(*
version 1.1		06. apr 2011
programmer		ks
tested by			ks

TN_SELECT_TEXT dient zur verwaltung und darstellung einer Elementeauswahl
*)
(* Benutzereingabe auswerten -> Selektion Text n *)
IF Xus_TN_INPUT_CONTROL_DATA.bo_Focus = TRUE THEN

(* Leertaste-Taste auswerten *)
	IF Xus_TN_INPUT_CONTROL_DATA.by_Input_ASCII_Code = BYTE#32 THEN
		Xus_TN_INPUT_CONTROL_DATA.in_selected := Xus_TN_INPUT_CONTROL_DATA.in_selected + INT#01; 
		Xus_TN_INPUT_CONTROL_DATA.bo_Update_Input := TRUE;
	END_IF;
 
	(* Return-Taste auswerten *)
	IF Xus_TN_INPUT_CONTROL_DATA.by_Input_Exten_Code = BYTE#13 THEN
		Xus_TN_INPUT_CONTROL_DATA.bo_Input_Entered := TRUE;
	END_IF;

END_IF;

(* Aktualisierung der Anzeige *)
IF (Xus_TN_INPUT_CONTROL_DATA.bo_Update_Input = TRUE) OR (Xus_TN_INPUT_CONTROL_DATA.bo_Update_All = TRUE) THEN

	(* Title-Text ausgeben *)
	IF Xus_TN_INPUT_CONTROL_DATA.bo_Update_All = TRUE THEN

		IF (Xus_TN_INPUT_CONTROL_DATA.in_Title_X_Offset = INT#00) AND (Xus_TN_INPUT_CONTROL_DATA.in_Title_Y_Offset = INT#00) THEN
			(* wenn Offset X,Y =0 dann Titlestring links vom Element positionieren *)
			FB_TN_SC_WRITE.Iin_Y := Xus_TN_INPUT_CONTROL_DATA.in_Y;
			FB_TN_SC_WRITE.Iin_X := Xus_TN_INPUT_CONTROL_DATA.in_X - LEN(Xus_TN_INPUT_CONTROL_DATA.st_Title_String);

		ELSE
			(* Title-Text durch Row, Color-Offset ausgeben *)
			FB_TN_SC_WRITE.Iin_Y := Xus_TN_INPUT_CONTROL_DATA.in_Y + Xus_TN_INPUT_CONTROL_DATA.in_Title_Y_Offset;
			FB_TN_SC_WRITE.Iin_X := Xus_TN_INPUT_CONTROL_DATA.in_X + Xus_TN_INPUT_CONTROL_DATA.in_Title_X_Offset;
		END_IF;

		(* Title-Text durch Row, Color-Offset ausgeben *)
		FB_TN_SC_WRITE(	Iby_ATTR := Xus_TN_INPUT_CONTROL_DATA.by_Title_Attr,
						Ist_STRING := Xus_TN_INPUT_CONTROL_DATA.st_Title_String,
						Xus_TN_SCREEN := Xus_TN_SCREEN);

	END_IF;

	(* Eingabezeile verarbeiten *)

	(* Anzahl der Elemente bestimmen *)
	in_count := ELEMENT_COUNT(SEP:=BYTE#35,ELEMENT:=Xus_TN_INPUT_CONTROL_DATA.st_Input_Data);

	IF in_Count > INT#00 THEN

		IF Xus_TN_INPUT_CONTROL_DATA.in_selected < INT#1 THEN
			Xus_TN_INPUT_CONTROL_DATA.in_selected := INT#01;
		END_IF;

		IF Xus_TN_INPUT_CONTROL_DATA.in_selected > in_count THEN
			Xus_TN_INPUT_CONTROL_DATA.in_selected := INT#01;
		END_IF;

		st_String := ELEMENT_GET(SEP:=BYTE#35,POS:=Xus_TN_INPUT_CONTROL_DATA.in_selected - 1,ELEMENT:=Xus_TN_INPUT_CONTROL_DATA.st_Input_Data);

		st_String := FIX(	str:=st_String,
							L:=LEN(Xus_TN_INPUT_CONTROL_DATA.st_Input_Mask),
							C:=BYTE#32,
							M:=Xus_TN_INPUT_CONTROL_DATA.in_Input_Option);

		Xus_TN_INPUT_CONTROL_DATA.st_Input_String := st_String;

		IF Xus_TN_INPUT_CONTROL_DATA.bo_Focus = TRUE THEN
			by_Attr := Xus_TN_INPUT_CONTROL_DATA.by_Attr_mF;
		ELSE
			by_Attr := Xus_TN_INPUT_CONTROL_DATA.by_Attr_oF;
		END_IF;

		FB_TN_SC_WRITE(	Iin_Y := Xus_TN_INPUT_CONTROL_DATA.in_Y,
						Iin_X := Xus_TN_INPUT_CONTROL_DATA.in_X,
						Iby_ATTR := by_Attr,
						Ist_STRING := st_String,
						Xus_TN_SCREEN := Xus_TN_SCREEN);
	END_IF;

	(* Cursor auf aktuelle Position setzen *)
	Xus_TN_INPUT_CONTROL_DATA.in_Cursor_Y := Xus_TN_INPUT_CONTROL_DATA.in_Y;
	Xus_TN_INPUT_CONTROL_DATA.in_Cursor_X := Xus_TN_INPUT_CONTROL_DATA.in_X;

	(* Update-Flag's rücksetzen *)
	Xus_TN_INPUT_CONTROL_DATA.bo_Update_All := FALSE;
	Xus_TN_INPUT_CONTROL_DATA.bo_Update_Input := FALSE;

END_IF;

(* revision history

ks	06. apr. 2011	rev 1.1
	list_len und list_get durch element_count und element_get ersetzt

ks	10. mai. 2010	rev 1.0
	original version
*)
END_FUNCTION_BLOCK

(* POU TN_INPUT_EDIT_LINE, ST *)
FUNCTION_BLOCK TN_INPUT_EDIT_LINE
VAR
	in_count : INT;
	in_Count_End : INT;
	in_CursorOffset : INT;
	by_Attr : BYTE;
	st_String : STRING;
	bo_Pos_Found : BOOL;
	st_CHAR : STRING(1);
	in_old_charpos : INT;
END_VAR
VAR
	FB_TN_SC_WRITE : TN_SC_WRITE;
END_VAR
VAR_IN_OUT
	Xus_TN_SCREEN : us_TN_SCREEN;
	Xus_TN_INPUT_CONTROL_DATA : us_TN_INPUT_CONTROL_DATA;
END_VAR

(*
version 1.0		10. mai 2010
programmer		ks
tested by		ks

TN_INPUT_EDIT_LINE ermöglicht die Eingabe von Texten durch eine Editierbare Eingabezeile
*)
(* Cursorsteuerung rücksetzen *)
in_CursorOffset := INT#0;

IF Xus_TN_INPUT_CONTROL_DATA.bo_Focus = TRUE THEN

	(* Texteingabe erkannt ? *)
	IF Xus_TN_INPUT_CONTROL_DATA.by_Input_ASCII_Code > BYTE#0 THEN

		IF (Xus_TN_INPUT_CONTROL_DATA.bo_Input_Only_Num = TRUE AND Xus_TN_INPUT_CONTROL_DATA.bo_Input_ASCII_IsNum = TRUE)
			OR (Xus_TN_INPUT_CONTROL_DATA.bo_Input_Only_Num = FALSE) THEN

			(* ASCII Wert in einen String wandeln *)
			st_CHAR := CHR_TO_STRING(C:=Xus_TN_INPUT_CONTROL_DATA.by_Input_ASCII_Code);

			(* Eingabe übernehmen *)
			Xus_TN_INPUT_CONTROL_DATA.st_Input_Data := REPLACE(Xus_TN_INPUT_CONTROL_DATA.st_Input_Data,
			st_CHAR,INT#1,Xus_TN_INPUT_CONTROL_DATA.in_Cursor_Pos);

			in_CursorOffset := INT#1;
			Xus_TN_INPUT_CONTROL_DATA.bo_Update_Input := TRUE;
		END_IF;
	END_IF;

	CASE BYTE_TO_INT(Xus_TN_INPUT_CONTROL_DATA.by_Input_Exten_Code) OF

	67: (* Cursor rechts gedrückt *)
		in_CursorOffset := INT#1;

	68: (* Cursor links gedrückt *)
		in_CursorOffset := -1;

	08: (* Backspace gedrückt *)
		Xus_TN_INPUT_CONTROL_DATA.st_Input_Data := REPLACE(Xus_TN_INPUT_CONTROL_DATA.st_Input_Data, ' ', 1,Xus_TN_INPUT_CONTROL_DATA.in_Cursor_Pos);
		Xus_TN_INPUT_CONTROL_DATA.bo_Update_Input := TRUE;
		in_CursorOffset := -1;

	13: (* Enter-Taste gedrückt *)
		IF LEN(Xus_TN_INPUT_CONTROL_DATA.st_Input_Mask) > INT#00 THEN
			(* Eingabestring übernehmen *)
			Xus_TN_INPUT_CONTROL_DATA.st_Input_String := Xus_TN_INPUT_CONTROL_DATA.st_Input_Data;

			(* Eingabestring -> links und rechts Leerzeichen entfernen *)
			Xus_TN_INPUT_CONTROL_DATA.st_Input_String := TRIME(str:=Xus_TN_INPUT_CONTROL_DATA.st_Input_String);
			Xus_TN_INPUT_CONTROL_DATA.bo_Input_Entered := TRUE;

			(* neue Eingabe vorbereiten *)
			Xus_TN_INPUT_CONTROL_DATA.st_Input_Data := Xus_TN_INPUT_CONTROL_DATA.st_Input_Mask;

			Xus_TN_INPUT_CONTROL_DATA.in_Cursor_Pos := INT#1;
			Xus_TN_INPUT_CONTROL_DATA.bo_Update_Input := TRUE;

			(* suche erstes Position in Eingabemaske *)
			st_CHAR := MID(Xus_TN_INPUT_CONTROL_DATA.st_Input_Mask,1,Xus_TN_INPUT_CONTROL_DATA.in_Cursor_Pos);
			IF st_CHAR <> ' ' THEN
				(* nächsten Eingabeposition suchen *)
				in_CursorOffset := INT#1;
			END_IF;
		END_IF;
	END_CASE;
END_IF;

(* Cursor richtung rechts bewegen                                   *)
IF (in_CursorOffset > INT#0) OR (Xus_TN_INPUT_CONTROL_DATA.in_Cursor_Pos = INT#0) THEN
	bo_Pos_Found := FALSE;

	in_Count := Xus_TN_INPUT_CONTROL_DATA.in_Cursor_Pos + INT#1;
	in_Count_End := LEN(Xus_TN_INPUT_CONTROL_DATA.st_Input_Mask);

	WHILE (in_count <= in_Count_End) AND (bo_Pos_Found = FALSE) DO

		st_CHAR := MID(Xus_TN_INPUT_CONTROL_DATA.st_Input_Mask,1,in_count);
		IF st_CHAR = ' ' THEN
			Xus_TN_INPUT_CONTROL_DATA.in_Cursor_Pos := in_count;
			Xus_TN_INPUT_CONTROL_DATA.bo_Update_Input := TRUE;
			bo_Pos_Found := TRUE;
		END_IF;

		in_count := in_count + INT#1;

	END_WHILE;
END_IF;

(* Cursor richtung links bewegen *)
IF in_CursorOffset < INT#0 THEN
	bo_Pos_Found := FALSE;

	in_Count     := Xus_TN_INPUT_CONTROL_DATA.in_Cursor_Pos - INT#01;
	in_Count_End := INT#1;

	WHILE (in_count >= in_Count_End) AND (bo_Pos_Found = FALSE) DO

		st_CHAR := MID(Xus_TN_INPUT_CONTROL_DATA.st_Input_Mask,1,in_count);
		IF st_CHAR = ' ' THEN
			Xus_TN_INPUT_CONTROL_DATA.in_Cursor_Pos := in_count;
			Xus_TN_INPUT_CONTROL_DATA.bo_Update_Input := TRUE;
			bo_Pos_Found := TRUE;
		END_IF;

		in_count := in_count - INT#1;
	END_WHILE;
END_IF;

(* maximale Cursorposition ? *)
IF Xus_TN_INPUT_CONTROL_DATA.in_Cursor_Pos > LEN(Xus_TN_INPUT_CONTROL_DATA.st_Input_Data) THEN
	Xus_TN_INPUT_CONTROL_DATA.in_Cursor_Pos := LEN(Xus_TN_INPUT_CONTROL_DATA.st_Input_Data);
	Xus_TN_INPUT_CONTROL_DATA.bo_Update_Input := TRUE;
END_IF;

(* minimale Cursorposition ? *)
IF Xus_TN_INPUT_CONTROL_DATA.in_Cursor_Pos < INT#1 THEN
	Xus_TN_INPUT_CONTROL_DATA.in_Cursor_Pos := INT#1;
	Xus_TN_INPUT_CONTROL_DATA.bo_Update_Input := TRUE;
END_IF;

(* Aktualisierung der Anzeige *)
IF (Xus_TN_INPUT_CONTROL_DATA.bo_Update_Input = TRUE) OR (Xus_TN_INPUT_CONTROL_DATA.bo_Update_All = TRUE) THEN

	(* Title-Text ausgeben *)
	IF (Xus_TN_INPUT_CONTROL_DATA.bo_Update_All = TRUE) THEN

		IF (Xus_TN_INPUT_CONTROL_DATA.in_Title_X_Offset = INT#00) AND (Xus_TN_INPUT_CONTROL_DATA.in_Title_Y_Offset = INT#00) THEN
			(* wenn Offset X,Y =0 dann Titlestring links vom Element positionieren *)
			FB_TN_SC_WRITE.Iin_Y := Xus_TN_INPUT_CONTROL_DATA.in_Y;
			FB_TN_SC_WRITE.Iin_X := Xus_TN_INPUT_CONTROL_DATA.in_X - LEN(Xus_TN_INPUT_CONTROL_DATA.st_Title_String);
		ELSE
			(* Title-Text durch Row, Color-Offset ausgeben *)
			FB_TN_SC_WRITE.Iin_Y := Xus_TN_INPUT_CONTROL_DATA.in_Y + Xus_TN_INPUT_CONTROL_DATA.in_Title_Y_Offset;
			FB_TN_SC_WRITE.Iin_X := Xus_TN_INPUT_CONTROL_DATA.in_X + Xus_TN_INPUT_CONTROL_DATA.in_Title_X_Offset;
		END_IF;

		(* Title-Text durch Row, Color-Offset ausgeben *)
		FB_TN_SC_WRITE(	Iby_ATTR := Xus_TN_INPUT_CONTROL_DATA.by_Title_Attr,
						Ist_STRING := Xus_TN_INPUT_CONTROL_DATA.st_Title_String,
						Xus_TN_SCREEN := Xus_TN_SCREEN);
	END_IF;

	(* Eingabetext ausgeben *)
	IF (Xus_TN_INPUT_CONTROL_DATA.bo_Input_Hidden = TRUE) THEN

		st_String := '';

		IF LEN(Xus_TN_INPUT_CONTROL_DATA.st_Input_Data) = LEN(Xus_TN_INPUT_CONTROL_DATA.st_Input_Mask) THEN
			(* Eingabemodus: HIDDEN *)
			FOR in_count := 1 TO LEN(Xus_TN_INPUT_CONTROL_DATA.st_Input_Data) DO

				(* Zeichen aus Eingabemaske lesen *)
				st_CHAR := MID(Xus_TN_INPUT_CONTROL_DATA.st_Input_Mask,1,in_count);

				(* Eingabe oder Maskenzeichen ausgeben *)
				IF st_CHAR = ' ' THEN

					(* Zeichen aus Eingabedata lesen *)
					st_CHAR := MID(Xus_TN_INPUT_CONTROL_DATA.st_Input_Data,1,in_count);

					IF st_CHAR = ' ' THEN
						(* Leerzeichen ausgeben *)
						st_String := CONCAT(st_String, ' ');

					ELSE
						(* verdecktes Zeichen ausgeben *)
						st_String := CONCAT(st_String, '*');

					END_IF;

				ELSE
					(* Zeichen aus Eingabemaske übernehmen *)
					st_CHAR := MID(Xus_TN_INPUT_CONTROL_DATA.st_Input_Data,1,in_count);
					st_String := CONCAT(st_String,st_CHAR);

				END_IF;
			END_FOR;
		END_IF;
	ELSE

		(* Eingabemodus: NORMAL *)
		st_String := Xus_TN_INPUT_CONTROL_DATA.st_Input_Data;

	END_IF;

	(* String ausgeben *)

	IF Xus_TN_INPUT_CONTROL_DATA.bo_Focus = TRUE THEN
		by_Attr := Xus_TN_INPUT_CONTROL_DATA.by_Attr_mF;
	ELSE
		by_Attr := Xus_TN_INPUT_CONTROL_DATA.by_Attr_oF;
	END_IF;

	FB_TN_SC_WRITE(	Iin_Y := Xus_TN_INPUT_CONTROL_DATA.in_Y,
					Iin_X := Xus_TN_INPUT_CONTROL_DATA.in_X,
					Iby_ATTR := by_Attr,
					Ist_STRING := st_String,
					Xus_TN_SCREEN := Xus_TN_SCREEN);

	(* Cursor auf aktuelle Position setzen *)
	Xus_TN_INPUT_CONTROL_DATA.in_Cursor_Y := Xus_TN_INPUT_CONTROL_DATA.in_Y;
	Xus_TN_INPUT_CONTROL_DATA.in_Cursor_X := Xus_TN_INPUT_CONTROL_DATA.in_X + Xus_TN_INPUT_CONTROL_DATA.in_Cursor_Pos - INT#1;

	in_old_charpos := INT#0;

	(* Update-Flag's rücksetzen *)
	Xus_TN_INPUT_CONTROL_DATA.bo_Update_All := FALSE;
	Xus_TN_INPUT_CONTROL_DATA.bo_Update_Input := FALSE;
END_IF;

(* revision history
ks	10. mai. 2010	rev 1.0
	original version
*)
END_FUNCTION_BLOCK

(* POU TN_INPUT_MENU_BAR, ST *)
FUNCTION_BLOCK TN_INPUT_MENU_BAR
VAR
	FB_TN_INPUT_MENU_POPUP : TN_INPUT_MENU_POPUP;
	us_TN_MENU_POPUP : us_TN_MENU_POPUP;
	FB_TN_SC_WRITE_C : TN_SC_WRITE_C;
END_VAR
VAR
	in_ROW : INT;
	in_COL : INT;
	in_TITLE_Length : INT;
	st_MENU_BAR : STRING(STRING_LENGTH);
	st_MENU_TITLE : STRING;
	in_Count : INT;
	in_Index : INT;
	by_New_KeyCode : BYTE;
	in_Scroll_Offset : INT;
	by_ATTR : BYTE;
	bo_Reset_Position :	BOOL;
END_VAR
VAR_IN_OUT
	Xus_TN_MENU : us_TN_MENU;
	Xus_TN_SCREEN : us_TN_SCREEN;
END_VAR

(*
version 1.1		06. apr 2011
programmer		ks
tested by			ks

TN_MENU_BAR ermöglicht die verwaltung und darstellung einer MENU-BAR
*)
(* sicherstellen das rechteck immer innerhalb screen positioniert wird *)

IF (Xus_TN_MENU.in_State = INT#00) AND (Xus_TN_MENU.bo_Create = TRUE) THEN
	Xus_TN_MENU.in_State := INT#01;
	Xus_TN_MENU.bo_Create := FALSE;
	Xus_TN_MENU.in_Menu_Selected := INT#00;
	Xus_TN_MENU.bo_Update := TRUE;
	bo_Reset_Position := TRUE;

	(* Menu-Bar - Hauptmenue *)
	st_MENU_BAR := ELEMENT_GET(SEP:=BYTE#37,POS:=0,ELEMENT:=Xus_TN_MENU.st_MENU_TEXT);

	(* Menu-Bar - Anzahl der Elemente bestimmen *)
	Xus_TN_MENU.in_Menu_E_Count := ELEMENT_COUNT(SEP:=BYTE#35,ELEMENT:=st_MENU_BAR);

END_IF;

(* Keycode ablegen *)
by_New_KeyCode := Xus_TN_SCREEN.by_Input_Exten_Code;

(* Popup-Menu Tastensteuerung (nur Cursor oben + unten zulassen *)
IF (by_New_KeyCode = BYTE#65) OR (by_New_KeyCode = BYTE#66) THEN
	us_TN_MENU_POPUP.by_Input_Exten_Code := by_New_KeyCode;
ELSE
	us_TN_MENU_POPUP.by_Input_Exten_Code := BYTE#00;
END_IF;

(* Escape *)
IF (by_New_KeyCode = BYTE#27) THEN
	(* Menu war inaktiv -> Escape -> Menu aktivieren *)
	IF (Xus_TN_MENU.in_State = INT#01) AND (Xus_TN_SCREEN.bo_Modal_Dialog = FALSE) THEN
		Xus_TN_MENU.in_State := INT#02;
		Xus_TN_MENU.bo_Update := TRUE;
		Xus_TN_MENU.in_Menu_Selected := INT#00;

		Xus_TN_SCREEN.bo_Menue_Bar_Dialog := TRUE;

		(* Menu war aktiv -> Escape -> Menu deaktivieren *)
	ELSIF (Xus_TN_MENU.in_State = INT#02) THEN
		us_TN_MENU_POPUP.bo_Destroy := TRUE;
		Xus_TN_MENU.bo_Update := TRUE;
		Xus_TN_MENU.in_State := INT#01;
		bo_Reset_Position := TRUE;

		Xus_TN_SCREEN.bo_Menue_Bar_Dialog := FALSE;
	END_IF;
END_IF;

(* Menu aktiv *)
IF (Xus_TN_MENU.in_State = INT#02) THEN

	(* Return *)
	IF (by_New_KeyCode = BYTE#13)  THEN
		us_TN_MENU_POPUP.bo_Destroy := TRUE;
		Xus_TN_MENU.bo_Update := TRUE;
		Xus_TN_MENU.in_State := INT#01;
		bo_Reset_Position := TRUE;
		Xus_TN_MENU.in_Menu_Selected := (Xus_TN_MENU.in_Cur_Menu_Item * INT#10) + Xus_TN_MENU.in_Cur_Sub_Item;
		Xus_TN_SCREEN.by_Input_Exten_Code := BYTE#00;

		Xus_TN_SCREEN.bo_Menue_Bar_Dialog := FALSE;

		(* Destroy-Befehl -> Popup-Menu beenden *)
	ELSIF (Xus_TN_MENU.bo_Destroy = TRUE) THEN
		us_TN_MENU_POPUP.bo_Destroy := TRUE;
		Xus_TN_MENU.bo_Update := TRUE;
		Xus_TN_MENU.in_State := INT#01;
		bo_Reset_Position := TRUE;
		Xus_TN_MENU.in_Menu_Selected := INT#00;
		Xus_TN_SCREEN.by_Input_Exten_Code := BYTE#00;

		Xus_TN_SCREEN.bo_Menue_Bar_Dialog := FALSE;

	END_IF;

	IF (by_New_KeyCode = BYTE#67) THEN (* Cursor rechts *)
		in_Scroll_Offset := INT#1;
		Xus_TN_MENU.bo_Update := TRUE;
		Xus_TN_SCREEN.by_Input_Exten_Code := BYTE#00;

	ELSIF (by_New_KeyCode = BYTE#68) THEN (* Cursor links *)
		in_Scroll_Offset := -1;
		Xus_TN_MENU.bo_Update := TRUE;
		Xus_TN_SCREEN.by_Input_Exten_Code := BYTE#00;
	END_IF;
END_IF;

IF bo_Reset_Position = TRUE THEN
	bo_Reset_Position := FALSE;
	Xus_TN_MENU.in_X_SM_old := -1;
	Xus_TN_MENU.in_Y_SM_old := -1;
	Xus_TN_MENU.in_X_SM_new := -1;
	Xus_TN_MENU.in_Y_SM_new := -1;
END_IF;

(* POPUP-Menu updaten *)
IF (Xus_TN_MENU.in_State > INT#00) AND (Xus_TN_MENU.bo_Update = TRUE) THEN

	Xus_TN_MENU.bo_Update := FALSE; 

	in_ROW := Xus_TN_MENU.in_Y;
	in_COL := Xus_TN_MENU.in_X;

	(* Scrolloffset *)
	IF in_Scroll_Offset <> INT#00 THEN
		Xus_TN_MENU.in_Cur_Menu_Item := INC2(Xus_TN_MENU.in_Cur_Menu_Item,in_Scroll_Offset,1,Xus_TN_MENU.in_Menu_E_Count);
		in_Scroll_Offset := INT#00;
	ELSE
		(* Item = 0 und kein Scrolloffset *)
		IF (Xus_TN_MENU.in_Cur_Menu_Item = INT#00) THEN
			Xus_TN_MENU.in_Cur_Menu_Item := INT#01;
		END_IF;
	END_IF;

	(* alle Menutext zeichnen *)
	FOR in_Count := INT#01 TO Xus_TN_MENU.in_Menu_E_Count DO;

		(* Zeichenfarbe bestimmen *)
		IF (in_Count = Xus_TN_MENU.in_Cur_Menu_Item) AND (Xus_TN_MENU.in_State > INT#01 ) THEN
			by_ATTR := Xus_TN_MENU.by_Attr_mF;

			Xus_TN_MENU.in_Y_SM_new := in_ROW + INT#01;
			Xus_TN_MENU.in_X_SM_new := in_COL;

		ELSE
			by_ATTR := Xus_TN_MENU.by_Attr_oF;
		END_IF;

		st_MENU_TITLE := ELEMENT_GET(SEP:=BYTE#35,POS:=in_Count - 1,ELEMENT:=st_MENU_BAR);

		in_TITLE_Length := LEN(st_MENU_TITLE) + INT#02;

		FB_TN_SC_WRITE_C(	Iin_Y := in_ROW,
							Iin_X := in_COL,
							Iby_ATTR := by_ATTR,
							Iin_LENGTH := in_TITLE_Length,
							Iin_OPTION := INT#02,
							Ist_STRING := st_MENU_TITLE,
							Xus_TN_SCREEN := Xus_TN_SCREEN);

		in_COL := in_COL + in_TITLE_Length;

	END_FOR;
END_IF;

IF Xus_TN_MENU.in_X_SM_new <> Xus_TN_MENU.in_X_SM_old THEN

	(* SubMenu ist aktiv -> beenden                                     *)
	IF us_TN_MENU_POPUP.bo_Activ = TRUE THEN
		us_TN_MENU_POPUP.bo_Destroy := TRUE;

		(* Sub-Menu bearbeiten *)
		FB_TN_INPUT_MENU_POPUP(	Xus_TN_MENU_POPUP := us_TN_MENU_POPUP,
								Xus_TN_SCREEN := Xus_TN_SCREEN);
	END_IF;

	IF us_TN_MENU_POPUP.bo_Activ = FALSE THEN
		(* Popup-Menu zu aktuellen Menu parametrieren und ausführen         *)
		in_Index := Xus_TN_MENU.in_Cur_Menu_Item;

		us_TN_MENU_POPUP.in_Y := Xus_TN_MENU.in_Y_SM_new;
		us_TN_MENU_POPUP.in_X := Xus_TN_MENU.in_X_SM_new;
		us_TN_MENU_POPUP.by_Attr_mF := Xus_TN_MENU.by_Attr_mF;
		us_TN_MENU_POPUP.by_Attr_oF := Xus_TN_MENU.by_Attr_oF;
		us_TN_MENU_POPUP.st_Menu_Text := ELEMENT_GET(SEP:=BYTE#37,POS:=in_Index,ELEMENT:=Xus_TN_MENU.st_MENU_TEXT);
		us_TN_MENU_POPUP.bo_Create := TRUE;

		Xus_TN_MENU.in_X_SM_old := Xus_TN_MENU.in_X_SM_new;
		Xus_TN_MENU.in_Y_SM_old := Xus_TN_MENU.in_Y_SM_new;

	END_IF;
END_IF;

(* Popup-Menu zyklisch aufrufen *)
FB_TN_INPUT_MENU_POPUP(	Xus_TN_MENU_POPUP := us_TN_MENU_POPUP,
						Xus_TN_SCREEN := Xus_TN_SCREEN);

(* aktuelles Item vom Popup-Menu kopieren *)
Xus_TN_MENU.in_Cur_Sub_Item := us_TN_MENU_POPUP.in_Cur_Item;

(* Destroy-Befehl *)
IF (Xus_TN_MENU.in_State = INT#01) THEN
	IF (Xus_TN_MENU.bo_Destroy = TRUE) THEN
		Xus_TN_MENU.in_State := INT#00;
		Xus_TN_MENU.bo_Destroy := FALSE;
		Xus_TN_MENU.in_Cur_Menu_Item := INT#00;
		Xus_TN_MENU.in_Cur_Sub_Item := INT#00;
	END_IF;
END_IF;

(* revision history
ks	06. apr. 2011	rev 1.1
	list_len und list_get durch element_count und element_get ersetzt

ks	10. mai. 2010	rev 1.0
	original version
*)
END_FUNCTION_BLOCK

(* POU TN_RECEIVE, ST *)
FUNCTION_BLOCK TN_RECEIVE
VAR_IN_OUT
	R_BUF :	NETWORK_BUFFER;
	Xus_TN_SCREEN : us_TN_SCREEN;
END_VAR
VAR
	REQ_Size : UINT;
	REQ1 : BYTE;
	REQ2 : BYTE;
	REQ3 : BYTE;
END_VAR

(*
version 1.0		10. mai 2010
programmer		ks
tested by		ks

TN_RECEIVE empfängt Tastatureingaben vom Telnet Client und wertet diese aus
*)
(* Datenempfang auswertung *)
Xus_TN_SCREEN.by_Input_ASCII_Code := BYTE#00;
Xus_TN_SCREEN.by_Input_Exten_Code := BYTE#00;

IF R_BUF.SIZE > UINT#0 THEN
	(* empfangene Daten auswerten *)
	REQ_Size := R_BUF.SIZE;
	REQ1 := R_BUF.BUFFER[0];
	REQ2 := R_BUF.BUFFER[1];
	REQ3 := R_BUF.BUFFER[2];

	IF REQ1 = BYTE#27 AND REQ_Size >= UINT#3 THEN (* Escape *)
		IF REQ2 = BYTE#91 THEN (* Cursor code *)
			IF (REQ3 >= BYTE#65 AND REQ3 <= BYTE#68) OR (REQ3 = BYTE#72) OR (REQ3 = BYTE#75) THEN (* 65..68 = Cursor o,u,r,l / 72 = POS1 / 75 = ENDE *)
				Xus_TN_SCREEN.by_Input_Exten_Code := REQ3;
			END_IF;
		ELSIF REQ2 = BYTE#79 THEN (* Sondertasten F1/F2/F3/F4 *)
			IF REQ3 >= BYTE#80 AND REQ3 <= BYTE#83 THEN
				Xus_TN_SCREEN.by_Input_Exten_Code := REQ3;
			END_IF;
		END_IF;
	ELSIF REQ1 >= BYTE#32 AND REQ1 <= BYTE#126 THEN
		Xus_TN_SCREEN.by_Input_ASCII_Code := REQ1;
		Xus_TN_SCREEN.bo_Input_ASCII_IsNum := ISC_NUM(REQ1); (* Auswertung auf Zahleneingabe *)
	ELSIF REQ1 = BYTE#8 OR REQ1 = BYTE#9 OR REQ1 = BYTE#13 OR REQ1 = BYTE#27 THEN (* prüfe auf Steuerzeichen 8=Backspace / 9=Tabulator / 13=Return / 27=Escape *)
		Xus_TN_SCREEN.by_Input_Exten_Code := REQ1;
	END_IF;

	(* Empfangsbuffer Datenlänge null eintragen (Telegramm zerstören *)
	R_BUF.SIZE := UINT#00;
END_IF;

(* revision history
ks	10. mai. 2010	rev 1.0
	original version
*)
END_FUNCTION_BLOCK

(* POU TN_SEND_ROWS, ST *)
FUNCTION_BLOCK TN_SEND_ROWS
VAR_IN_OUT
	IP_C : IP_C;
	S_BUF : NETWORK_BUFFER;
	Xus_TN_SCREEN : us_TN_SCREEN;
END_VAR
VAR_INPUT
	S_BUF_SIZE : INT;
END_VAR
VAR
	in_Line_Count : INT;(*Zähler um max alle 24 Zeilen zu durchlaufen*)
	in_Col_Count : INT;
	in_Last_Row_Index : INT;
	bo_Break_Loop : BOOL;
	in_Row_Count : INT;
	in_Offset : INT;
	in_Write_Index : INT;
	in_Write_Index_Backup : INT;
	by_Cur_Color : BYTE;
	by_last_Color : BYTE;
	in_Write_Stop : INT;
END_VAR

(*
version 1.0		10. mai 2010
programmer		ks
tested by		ks

TN_SEND_ROWS prüft den Bildschirmspeicher auf änderungen, und sendet diese zeilenweise an den Telnet Client 
*)
(* Verbindung vorhanden und kein Datensenden aktiv *)
IF (IP_C.C_STATE < BYTE#127 OR S_BUF.SIZE > UINT#0) THEN
	RETURN; (* nein -> Baustein beenden *)
END_IF;

(* aktuellen Schreibindex laden *)
in_Write_Index := UINT_TO_INT(S_BUF.SIZE) - 1;

(* aktuellen Schreibindex zwischenspeichern *)
in_Write_Index_Backup := in_Write_Index;

(* positive Flanke Connect on *)
IF (IP_C.C_STATE = BYTE#254) OR (Xus_TN_SCREEN.bo_Clear_Screen) THEN

	(* Clear-Screen Meldung rücksetzen *)
	Xus_TN_SCREEN.bo_Clear_Screen := FALSE;

	(* alle Zeilen für Update markieren *)
	FOR in_Line_Count := INT#00 TO INT#23 DO
		Xus_TN_SCREEN.bya_Line_Update[in_Line_Count] := TRUE;
	END_FOR;

	(* ESC [0;30,40m  Reset Attributes + Black,Black *)
	in_Write_Index := in_Write_Index + INT#1;
	S_BUF.BUFFER[in_Write_Index] := BYTE#16#1B; (* ESC *)
	in_Write_Index := in_Write_Index + INT#1;
	S_BUF.BUFFER[in_Write_Index] := BYTE#16#5B; (* [ *)
	in_Write_Index := in_Write_Index + INT#1;
	S_BUF.BUFFER[in_Write_Index] := BYTE#16#30; (* 0 *)
	in_Write_Index := in_Write_Index + INT#1;
	S_BUF.BUFFER[in_Write_Index] := BYTE#16#3B; (* ; *)
	in_Write_Index := in_Write_Index + INT#1;
	S_BUF.BUFFER[in_Write_Index] := BYTE#16#33; (* 3 *)

	(* Einerstelle Farbe Foreground ausgeben *)
	in_Write_Index := in_Write_Index + INT#1;
	S_BUF.BUFFER[in_Write_Index] := (SHR(Xus_TN_SCREEN.by_Clear_Screen_Attr,4) OR BYTE#16#30);

	in_Write_Index := in_Write_Index + INT#1;
	S_BUF.BUFFER[in_Write_Index] := BYTE#16#3B; (* ; *)
	in_Write_Index := in_Write_Index + INT#1;
	S_BUF.BUFFER[in_Write_Index] := BYTE#16#34; (* 4 *)

	(* Einerstelle Farbe Background ausgeben *)
	in_Write_Index := in_Write_Index + INT#1;
	S_BUF.BUFFER[in_Write_Index] := ((Xus_TN_SCREEN.by_Clear_Screen_Attr AND BYTE#16#07) OR BYTE#16#30);

	in_Write_Index := in_Write_Index + INT#1;
	S_BUF.BUFFER[in_Write_Index] := BYTE#16#6D; (* m *)

	(* ESC[2J Clear screen and home cursor *)
	in_Write_Index := in_Write_Index + INT#1;
	S_BUF.BUFFER[in_Write_Index] := BYTE#16#1B; (* ESC *)
	in_Write_Index := in_Write_Index + INT#1;
	S_BUF.BUFFER[in_Write_Index] := BYTE#16#5B; (* [ *)
	in_Write_Index := in_Write_Index + INT#1;
	S_BUF.BUFFER[in_Write_Index] := BYTE#16#32; (* 2 *)
	in_Write_Index := in_Write_Index + INT#1;
	S_BUF.BUFFER[in_Write_Index] := BYTE#16#4A; (* J *)

	(* ESC [?7l Off *)
	in_Write_Index := in_Write_Index + INT#1;
	S_BUF.BUFFER[in_Write_Index] := BYTE#16#1B; (* ESC *)
	in_Write_Index := in_Write_Index + INT#1;
	S_BUF.BUFFER[in_Write_Index] := BYTE#16#5B; (* [ *)
	in_Write_Index := in_Write_Index + INT#1;
	S_BUF.BUFFER[in_Write_Index] := BYTE#16#3F; (* ? *)
	in_Write_Index := in_Write_Index + INT#1;
	S_BUF.BUFFER[in_Write_Index] := BYTE#16#37; (* 7 *)
	in_Write_Index := in_Write_Index + INT#1;
	S_BUF.BUFFER[in_Write_Index] := BYTE#16#6C; (* l *)

END_IF;

in_Last_Row_Index := INT#0;
bo_Break_Loop := FALSE;
in_Write_Stop := S_BUF_SIZE - 20;

(* alle Zeilen durchlaufen *)
FOR in_Line_Count := 0 TO 23 DO

	in_Offset := in_Row_Count * INT#80;

	(* prüfen ob Update einer Zeile notwendig ist bzw. nach Reconnect *)
	IF (Xus_TN_SCREEN.bya_Line_Update[in_Row_Count] = TRUE) THEN

		(* Schreib-Cursor positionieren *)
		in_Write_Index := in_Write_Index + INT#1;
		S_BUF.BUFFER[in_Write_Index] := BYTE#16#1B; (* ESC *)
		in_Write_Index := in_Write_Index + INT#1;
		S_BUF.BUFFER[in_Write_Index] := BYTE#16#5B; (* [ *)

		(* Zehnerstelle Zeilennummer ausgeben *)
		in_Write_Index := in_Write_Index + INT#1;
		S_BUF.BUFFER[in_Write_Index] :=
		SHR(INT_TO_BCDC(in_Row_Count + INT#1),INT#4) OR BYTE#16#30;

		(* Einerstelle Zeilennummer ausgeben *)
		in_Write_Index := in_Write_Index + INT#1;
		S_BUF.BUFFER[in_Write_Index] :=
		(INT_TO_BCDC(in_Row_Count + INT#1) AND BYTE#16#0F) OR BYTE#16#30;

		in_Write_Index := in_Write_Index + INT#1;
		S_BUF.BUFFER[in_Write_Index] := BYTE#16#3B; (* ; *)
		in_Write_Index := in_Write_Index + INT#1;
		S_BUF.BUFFER[in_Write_Index] := BYTE#16#31; (* 1 *)
		in_Write_Index := in_Write_Index + INT#1;
		S_BUF.BUFFER[in_Write_Index] := BYTE#16#48; (* H *)

		(* alle Spalten einer Zeile durchlaufen *)
		FOR in_Col_Count := 0 TO 79 DO

			(* aktuelle Farbe bestimmen *)
			by_Cur_Color := Xus_TN_SCREEN.bya_COLOR[in_Offset];
			IF (by_Cur_Color <> by_last_Color) OR (in_Col_Count = INT#00) THEN

				(* Farbeinstellung: ANSI-Sequenz ESC[X;Y;Zm ausgeben *)
				in_Write_Index := in_Write_Index + INT#1;
				S_BUF.BUFFER[in_Write_Index] := BYTE#16#1B; (* ESC *)

				in_Write_Index := in_Write_Index + INT#1;
				S_BUF.BUFFER[in_Write_Index] := BYTE#16#5B; (* [ *)

				(* Farbeinstellung: dunkel oder Hell und blinken bestimmen *)

					IF (((by_Cur_Color AND BYTE#2#10001000) XOR (by_last_Color AND BYTE#2#10001000)) <> BYTE#00) OR (in_Col_Count = 0) THEN

						in_Write_Index := in_Write_Index + INT#1;
						S_BUF.BUFFER[in_Write_Index] := BYTE#16#30; (* 0 *)
						in_Write_Index := in_Write_Index + INT#1;
						S_BUF.BUFFER[in_Write_Index] := BYTE#16#3B; (* ; *)

						(* keine dunklen Farben gewünscht -> dann Bold & Bright *)
						IF (by_Cur_Color AND BYTE#2#00001000) = BYTE#2#00000000 THEN

							(* auf Bold & Btight Farben umstellen *)
							in_Write_Index := in_Write_Index + INT#1;
							S_BUF.BUFFER[in_Write_Index] := BYTE#16#31; (* 1 *) 
							in_Write_Index := in_Write_Index + INT#1;
							S_BUF.BUFFER[in_Write_Index] := BYTE#16#3B; (* ; *)

						END_IF;

						(* blinkenden Farben gewünscht *)
						IF (by_Cur_Color AND BYTE#2#10000000) = BYTE#2#10000000 THEN 

							(* auf Bold & Bright Farben umstellen *)
							in_Write_Index := in_Write_Index + INT#1;
							S_BUF.BUFFER[in_Write_Index] := BYTE#16#35; (* 5 *) 
							in_Write_Index := in_Write_Index + INT#1;
							S_BUF.BUFFER[in_Write_Index] := BYTE#16#3B; (* ; *)

						END_IF;

					END_IF;

					(* Zehnerstelle Farbe Foreground ausgeben *)
					in_Write_Index := in_Write_Index + INT#1;
					S_BUF.BUFFER[in_Write_Index] := BYTE#16#33; (* 3 *)

					(* Einerstelle Farbe Foreground ausgeben *)
					in_Write_Index := in_Write_Index + INT#1;
					S_BUF.BUFFER[in_Write_Index] := ((SHR(by_Cur_Color,4) AND BYTE#2#00000111) OR BYTE#16#30);

					in_Write_Index := in_Write_Index + INT#1;
					S_BUF.BUFFER[in_Write_Index] := BYTE#16#3B; (* ; *)

					(* Zehnerstelle Farbe Background ausgeben *)
					in_Write_Index := in_Write_Index + INT#1;
					S_BUF.BUFFER[in_Write_Index] := BYTE#16#34; (* 4 *)

					(* Einerstelle Farbe Background ausgeben *)
					in_Write_Index := in_Write_Index + INT#1;
					S_BUF.BUFFER[in_Write_Index] := ((by_Cur_Color AND BYTE#2#00000111) OR BYTE#16#30); 

					in_Write_Index := in_Write_Index + INT#1;
					S_BUF.BUFFER[in_Write_Index] := BYTE#16#6D; (* m *)

					(* neue Farbe als letzt verwendete speichern *)
					by_last_Color := by_Cur_Color;

				END_IF;

				(* Buffer Ende vorzeitig erreicht -> Ende *)
				IF (in_Write_Index > in_Write_Stop) THEN

					bo_Break_Loop := TRUE;
					EXIT;

				END_IF;

				(* ein TEXT-Zeichen von Screenbuffer in den Sendebuffer übertragen *)
				in_Write_Index := in_Write_Index + INT#1;
				S_BUF.BUFFER[in_Write_Index] := Xus_TN_SCREEN.bya_CHAR[in_Offset];

				(* nächste Spalte anwählen *)
				in_Offset := in_Offset + INT#01;
			END_FOR;

			IF (bo_Break_Loop = TRUE) THEN;

				(* Buffer Ende vorzeitig erreicht -> nur bis zur letzten kompletten Zeile uebertragen *)
				in_Write_Index := in_Last_Row_Index;

				EXIT;
			END_IF;

			(* Buffer ist noch nicht voll -> neue Zeile ubernehmen *)
			in_Last_Row_Index := in_Write_Index;
			Xus_TN_SCREEN.bya_Line_Update[in_Row_Count] := FALSE;

		END_IF;

		(* naechste Zeile adressieren *)
		in_Row_Count := in_Row_Count + INT#01;

		(* ab letzter Zeile wieder von vorne beginnen *)
		IF (in_Row_Count > INT#23) THEN
			in_Row_Count := INT#00;
		END_IF;
		(*-----------------------------------------------*)


	END_FOR;

	(* wenn in einen Update-Zyklus alle Zeilen auf einmal geschafft wurden *)
	(* wird der Row_Count auf ersten Zeile gestellt *)
	(* soll das hässliche Grafikflackern verhindern *)
	(* ansonsten wird bei der letzen Zeile weitergemacht *)
	IF (bo_Break_Loop = FALSE) THEN
		in_Row_Count := INT#00;
	END_IF;

	(* Edit-Cursor positionieren *)
	IF (in_Write_Index <> in_Write_Index_Backup) THEN

		in_Write_Index := in_Write_Index + INT#1;
		S_BUF.BUFFER[in_Write_Index] := BYTE#16#1B; (* ESC *)
		in_Write_Index := in_Write_Index + INT#1;
		S_BUF.BUFFER[in_Write_Index] := BYTE#16#5B; (* [ *)

		(* Zehnerstelle Zeilennummer ausgeben *)
		in_Write_Index := in_Write_Index + INT#1;
		S_BUF.BUFFER[in_Write_Index] := SHR(INT_TO_BCDC(Xus_TN_SCREEN.in_Cursor_Y + 1),INT#4) OR BYTE#16#30;

		(* Einerstelle Zeilennummer ausgeben *)
		in_Write_Index := in_Write_Index + INT#1;
		S_BUF.BUFFER[in_Write_Index] := (INT_TO_BCDC(Xus_TN_SCREEN.in_Cursor_Y + 1) AND BYTE#16#0F) OR BYTE#16#30;

		in_Write_Index := in_Write_Index + INT#1;
		S_BUF.BUFFER[in_Write_Index] := BYTE#16#3B; (* ; *)

		(* Zehnerstelle Spaltenummer ausgeben *)
		in_Write_Index := in_Write_Index + INT#1;
		S_BUF.BUFFER[in_Write_Index] := SHR(INT_TO_BCDC(Xus_TN_SCREEN.in_Cursor_X + 1),INT#4) OR BYTE#16#30;

		(* Einerstelle Spaltennummer ausgeben *)
		in_Write_Index := in_Write_Index + INT#1;
		S_BUF.BUFFER[in_Write_Index] := (INT_TO_BCDC(Xus_TN_SCREEN.in_Cursor_X + 1) AND BYTE#16#0F) OR BYTE#16#30;

		in_Write_Index := in_Write_Index + INT#1;
		S_BUF.BUFFER[in_Write_Index] := BYTE#16#48; (* H *)

END_IF;

(* aktuellen Schreibindex speichern -> Senden anstossen *)
S_BUF.SIZE := INT_TO_UINT(in_Write_Index + 1);

(* revision history
ks	10. mai. 2010	rev 1.0
	original version
*)
END_FUNCTION_BLOCK

(* POU LOG_VIEWPORT, ST *)
FUNCTION_BLOCK LOG_VIEWPORT
VAR_IN_OUT
	LC : LOG_CONTROL;
	LV : us_LOG_VIEWPORT;
END_VAR
VAR
	pos : INT;
	count : INT;
	idx : INT;
	base : INT;
	update_pos : BOOL;
END_VAR

(*
version 1.0		01 mai 2010
programmer		ks
tested BY		ks

LOG_VIEWPORT erzeugt einen Liste der Meldungen des Loggingbuffers die innerhalb einer virtuellen Ansicht enthalten sind.
*)
(* Scroll Button verarbeiten *)
IF LV.MOVE_TO_X <> 0 THEN
	CASE LV.MOVE_TO_X OF
	30000: pos := 1 ; (* älteste Meldung anzeigen *)
	30001: pos := LC.SIZE; (* neueste Meldung anzeigen *)
	30002: pos := pos + LV.COUNT; (* eine Seite nach unten blättern -> Richtung neuere Nachrichten *)
	30003: pos := pos - LV.COUNT; (* eine Seite nach oben blättern -> Richtung ältere Nachrichten *)
	ELSE
		pos := pos + LV.MOVE_TO_X;
	END_CASE;
	update_pos := TRUE;
	LV.MOVE_TO_X := 0;
END_IF;

IF (LV.UPDATE_COUNT <> LC.UPDATE_COUNT) OR update_pos THEN (* Aktualisierung überwachen *)
	LV.UPDATE := TRUE;
	LV.UPDATE_COUNT := LC.UPDATE_COUNT;
	update_pos := FALSE;

	(* pos prüfen und übernehmen *)
	IF LC.RING_MODE THEN
		pos := LIMIT(1,pos,LC.SIZE - LV.COUNT + 1);
	ELSE
		IF LC.IDX > LV.COUNT THEN
			pos := LIMIT(1,pos,LC.IDX - LV.COUNT + 1);
		ELSE
			pos := 1;
		END_IF;
	END_IF;

	(* idxBasis berechnen *)
	base := LC.IDX - pos - LV.COUNT + 1;
	IF LC.RING_MODE THEN 
		(* Anzeige im Ringpuffermodus *)
		FOR count:= 1 TO LV.COUNT DO
			idx := base + count;
			IF idx < 1 THEN
				idx := idx + LC.SIZE;
			END_IF;
		END_FOR;
	ELSE
		(* Anzeige im Normalmodus *)
		FOR count:= 1 TO LV.COUNT DO
			idx := base + count;
			IF idx < 1 THEN
				(* Leere Zeile ausgeben *)
				LV.LINE_ARRAY[count] := 0;
			ELSE
				LV.LINE_ARRAY[count] := idx;
			END_IF;
		END_FOR;
	END_IF;
END_IF;

(* revision history
ks	01. mai 2010	rev 1.0
	original version
*)
END_FUNCTION_BLOCK

(* POU TN_SC_VIEWPORT, ST *)
FUNCTION_BLOCK TN_SC_VIEWPORT
VAR
	FB_TN_SC_WRITE : TN_SC_WRITE;
	FB_TON : TON;
END_VAR
VAR
	in_index : INT;
	in_Color : INT;
	by_Attr : BYTE;
	in_count : INT;
END_VAR
VAR_IN_OUT
	Xus_LOG_VIEWPORT : us_LOG_VIEWPORT;
	Xus_LOG_CONTROL : LOG_CONTROL;
	Xus_TN_SCREEN : us_TN_SCREEN;
END_VAR
VAR_INPUT
	Iin_X : INT;
	Iin_Y : INT;
	Iin_Width : INT;
	Idw_ATTR_1 : DWORD;
	Idw_ATTR_2 : DWORD;
	Iti_TIME : TIME;
END_VAR

(*
version 1.0		10. mai 2010
programmer		ks
tested by		ks

TN_SC_VIEWPORT verwaltet und zeichnet einen rechteckigen Bereich in dem der Log-buffer angezeigt wird
*)
(* LOG-Messages ausgeben *)

IF Xus_LOG_VIEWPORT.UPDATE AND FB_TON.Q THEN (* Update gewünscht und Verzögerungszeit abgelaufen *)
	Xus_LOG_VIEWPORT.UPDATE := FALSE;
	FOR in_count := 1 TO Xus_LOG_VIEWPORT.COUNT DO (* Alle Viewport-Zeilen abarbeiten *)
		in_index := Xus_LOG_VIEWPORT.LINE_ARRAY[in_count];
		(* Farbe aus den Option-Parameter auslesen >0,Level,Back,Front< *)
		in_Color := DWORD_TO_INT(Xus_LOG_CONTROL.MSG_OPTION[in_index] AND DWORD#2#1111);

		CASE in_Color OF
		0..3: by_Attr := BYTE_OF_DWORD(Idw_ATTR_1,INT_TO_BYTE(in_Color));
		4..7: by_Attr := BYTE_OF_DWORD(Idw_ATTR_2,INT_TO_BYTE(in_Color));
		ELSE
			by_Attr := BYTE_OF_DWORD(Idw_ATTR_1,BYTE#0);
		END_CASE;

		(* Message (Text + Farbe) ausgeben *)
		FB_TN_SC_WRITE(	Iin_Y := Iin_Y + in_count - INT#01,
						Iin_X := Iin_X,
						Iby_ATTR := by_Attr,
						Ist_STRING := FIX(str := Xus_LOG_CONTROL.MSG[in_index], L := Iin_Width, C := BYTE#32, M := INT#00), (* String rechts ergänzen bzw. kürzen *)
						Xus_TN_SCREEN := Xus_TN_SCREEN);

	END_FOR;

	(* Timer stoppen/rücksetzen *)
	FB_TON.IN := FALSE;
	FB_TON.PT := Iti_TIME;
	FB_TON();

END_IF;

(* Update-Zeitverzoegerung *)
FB_TON.IN := TRUE;
FB_TON.PT := Iti_TIME;
FB_TON();

(* revision history
ks	10. mai. 2010	rev 1.0
	original version
*)
END_FUNCTION_BLOCK

(* POU TN_VISION_DEMO_2, ST *)
PROGRAM TN_VISION_DEMO_2
VAR
	FB_TN_FRAMEWORK : TN_FRAMEWORK;
	FB_TN_SC_FILL : TN_SC_FILL;
	FB_TN_SC_WRITE_C : TN_SC_WRITE_C;
	FB_TN_SC_WRITE : TN_SC_WRITE;
	Xus_TN_MENU : us_TN_MENU;
	Xus_TN_INPUT_CONTROL : us_TN_INPUT_CONTROL;
	Xus_TN_SCREEN : us_TN_SCREEN;
	S_BUF : NETWORK_BUFFER;
	R_BUF : NETWORK_BUFFER;
	IP_C : IP_C;
END_VAR
FB_TN_FRAMEWORK(
	us_TN_INPUT_CONTROL := Xus_TN_INPUT_CONTROL ,
	us_TN_SCREEN := Xus_TN_SCREEN ,
	us_TN_MENU := Xus_TN_MENU ,
	S_BUF := S_BUF ,
	R_BUF:= R_BUF ,
	IP_C:= IP_C );

(* Initialisierung der Daten und Strukturen *)
IF (Xus_TN_SCREEN.in_Page_Number = INT#00) THEN
	Xus_TN_SCREEN.in_Page_Number := INT#01;

	(* Clear-Screen (Farbe setzen + Display löschen) *)
	Xus_TN_SCREEN.by_Clear_Screen_Attr := BYTE#16#00;
	Xus_TN_SCREEN.bo_Clear_Screen := TRUE;

	(* Screen initialisieren (mit Leerzeichen füllen) *)
	FB_TN_SC_FILL(	Iin_X1 := INT#00,
					Iin_Y1 := INT#00,
					Iin_X2 := INT#79,
					Iin_Y2 := INT#23,
					Iby_CHAR := BYTE#32,
					Iby_Attr := BYTE#16#00,
					Xus_TN_SCREEN := Xus_TN_SCREEN);

	(* Statische Texte ausgeben *)
	FB_TN_SC_WRITE(	Iin_X := INT#00,
					Iin_Y := INT#00,
					Iby_ATTR := BYTE#16#70,
					Ist_STRING := 'Login Screen                                                     FL SWITCH MM HS',
					Xus_TN_SCREEN := Xus_TN_SCREEN);

	(* Statische Texte ausgeben *)
	FB_TN_SC_WRITE(	Iin_X := INT#00,
					Iin_Y := INT#03,
					Iby_ATTR := BYTE#16#70,
					Ist_STRING := 'XXXXXXXXX',
					Xus_TN_SCREEN := Xus_TN_SCREEN);

	(* Statische Texte ausgeben *)
	FB_TN_SC_WRITE(	Iin_X := INT#00,
					Iin_Y := INT#04,
					Iby_ATTR := BYTE#16#70,
					Ist_STRING := 'X   X  XX',
					Xus_TN_SCREEN := Xus_TN_SCREEN);

	(* Statische Texte ausgeben *)
	FB_TN_SC_WRITE(	Iin_X := INT#00,
					Iin_Y := INT#05,
					Iby_ATTR := BYTE#16#70,
					Ist_STRING := 'X   O   X      ---> Phoenix Contact Managed Switch System <---',
					Xus_TN_SCREEN := Xus_TN_SCREEN);

	(* Statische Texte ausgeben *)
	FB_TN_SC_WRITE(	Iin_X := INT#00,
					Iin_Y := INT#06,
					Iby_ATTR := BYTE#16#70,
					Ist_STRING := 'X   X  XX               Phoenix Contact GmbH & Co KG',
					Xus_TN_SCREEN := Xus_TN_SCREEN);

	(* Statische Texte ausgeben *)
	FB_TN_SC_WRITE(	Iin_X := INT#00,
					Iin_Y := INT#07,
					Iby_ATTR := BYTE#16#70,
					Ist_STRING := 'X   XXXXX                   www.PhoenixContact.com',
					Xus_TN_SCREEN := Xus_TN_SCREEN);

	(* Statische Texte ausgeben *)
	FB_TN_SC_WRITE(	Iin_X := INT#00,
					Iin_Y := INT#08,
					Iby_ATTR := BYTE#16#70,
					Ist_STRING := 'X   XXXXX',
					Xus_TN_SCREEN := Xus_TN_SCREEN);

	(* Statische Texte ausgeben *)
	FB_TN_SC_WRITE(	Iin_X := INT#00,
					Iin_Y := INT#09,
					Iby_ATTR := BYTE#16#70,
					Ist_STRING := 'XXXXXXXXX',
					Xus_TN_SCREEN := Xus_TN_SCREEN);

	(* Statische Texte ausgeben *)
	FB_TN_SC_WRITE(	Iin_X := INT#00,
					Iin_Y := INT#11,
					Iby_ATTR := BYTE#16#70,
					Ist_STRING := '                Running switch application version:  4.00',
					Xus_TN_SCREEN := Xus_TN_SCREEN);

	(* Alle Input-Controls initialisieren *)

	Xus_TN_INPUT_CONTROL.bo_Enable := FALSE;

  (* Initialisierung der Eingabe-Zeile *)
	Xus_TN_INPUT_CONTROL.usa_TN_INPUT_CONTROL_DATA[1].in_Type := INT#01;
	Xus_TN_INPUT_CONTROL.usa_TN_INPUT_CONTROL_DATA[1].in_Y := INT#17;
	Xus_TN_INPUT_CONTROL.usa_TN_INPUT_CONTROL_DATA[1].in_X := INT#33;
	Xus_TN_INPUT_CONTROL.usa_TN_INPUT_CONTROL_DATA[1].by_Attr_mF := BYTE#16#70;
	Xus_TN_INPUT_CONTROL.usa_TN_INPUT_CONTROL_DATA[1].by_Attr_oF := BYTE#16#70;
	Xus_TN_INPUT_CONTROL.usa_TN_INPUT_CONTROL_DATA[1].in_Cursor_Pos := INT#0;
	Xus_TN_INPUT_CONTROL.usa_TN_INPUT_CONTROL_DATA[1].bo_Input_Only_Num := FALSE;
	Xus_TN_INPUT_CONTROL.usa_TN_INPUT_CONTROL_DATA[1].bo_Input_Hidden := TRUE;
	Xus_TN_INPUT_CONTROL.usa_TN_INPUT_CONTROL_DATA[1].st_Input_Mask := '                ';
	Xus_TN_INPUT_CONTROL.usa_TN_INPUT_CONTROL_DATA[1].st_Input_Data := Xus_TN_INPUT_CONTROL.usa_TN_INPUT_CONTROL_DATA[1].st_Input_Mask;
	Xus_TN_INPUT_CONTROL.usa_TN_INPUT_CONTROL_DATA[1].st_Input_ToolTip := '';
	Xus_TN_INPUT_CONTROL.usa_TN_INPUT_CONTROL_DATA[1].in_Input_Option := INT#00;
	Xus_TN_INPUT_CONTROL.usa_TN_INPUT_CONTROL_DATA[1].in_Title_Y_Offset := INT#00;
	Xus_TN_INPUT_CONTROL.usa_TN_INPUT_CONTROL_DATA[1].in_Title_X_Offset := -12;
	Xus_TN_INPUT_CONTROL.usa_TN_INPUT_CONTROL_DATA[1].by_Title_Attr := BYTE#16#70;
	Xus_TN_INPUT_CONTROL.usa_TN_INPUT_CONTROL_DATA[1].st_Title_String := 'Password:  [                ]';

	(* Control-Tool-Tip *)
	Xus_TN_INPUT_CONTROL.in_ToolTip_Y := INT#23;
	Xus_TN_INPUT_CONTROL.in_ToolTip_X := INT#09;
	Xus_TN_INPUT_CONTROL.by_ToolTip_Attr := BYTE#16#70;
	Xus_TN_INPUT_CONTROL.in_ToolTip_Size := INT#30;

	(* Control-Verwaltung initialisieren *)
	Xus_TN_INPUT_CONTROL.in_Count := INT#01;
	Xus_TN_INPUT_CONTROL.bo_Enable := TRUE;
	Xus_TN_INPUT_CONTROL.bo_Reset_Fokus := TRUE;
END_IF;

IF (Xus_TN_SCREEN.in_Page_Number = INT#01) THEN

	(* eingegebenen String übernehmen *)
	IF Xus_TN_INPUT_CONTROL.usa_TN_INPUT_CONTROL_DATA[1].bo_Input_Entered = TRUE THEN

		Xus_TN_INPUT_CONTROL.usa_TN_INPUT_CONTROL_DATA[1].bo_Input_Entered := FALSE;

		Xus_TN_INPUT_CONTROL.usa_TN_INPUT_CONTROL_DATA[1].st_Input_String :=
			LOWERCASE(str:=Xus_TN_INPUT_CONTROL.usa_TN_INPUT_CONTROL_DATA[1].st_Input_String);

		IF Xus_TN_INPUT_CONTROL.usa_TN_INPUT_CONTROL_DATA[1].st_Input_String = 'oscat' THEN
			Xus_TN_SCREEN.in_Page_Number := INT#04;

		ELSE
			FB_TN_SC_WRITE_C(	Iin_Y := Xus_TN_INPUT_CONTROL.in_ToolTip_Y,
								Iin_X := Xus_TN_INPUT_CONTROL.in_ToolTip_X,
								Iby_ATTR := BYTE#16#F1,
								Iin_OPTION := INT#02, (* Center-String *)
								Iin_LENGTH := Xus_TN_INPUT_CONTROL.in_ToolTip_Size,
								Ist_STRING := ' User Password Failed   ',
								Xus_TN_SCREEN := Xus_TN_SCREEN);
		END_IF;
	END_IF;
END_IF;

(* Initialisierung der Daten und Strukturen *)
IF (Xus_TN_SCREEN.in_Page_Number = INT#04) THEN
	Xus_TN_SCREEN.in_Page_Number := INT#05;

	(* Clear-Screen (Farbe setzen + Display löschen) *)
	Xus_TN_SCREEN.by_Clear_Screen_Attr := BYTE#16#00;
	Xus_TN_SCREEN.bo_Clear_Screen := TRUE;

	(* Screen initialisieren (mit Leerzeichen füllen) *)
	FB_TN_SC_FILL(	Iin_X1 := INT#00,
					Iin_Y1 := INT#00,
					Iin_X2 := INT#79,
					Iin_Y2 := INT#23,
					Iby_CHAR := BYTE#32,
					Iby_Attr := BYTE#16#00,
					Xus_TN_SCREEN := Xus_TN_SCREEN);

	(* Statische Texte ausgeben *)
	FB_TN_SC_WRITE(	Iin_X := INT#00,
					Iin_Y := INT#00,
					Iby_ATTR := BYTE#16#70,
					Ist_STRING := 'Basic Switch Configuration                                       FL SWITCH MM HS',
					Xus_TN_SCREEN := Xus_TN_SCREEN);

	(* Statische Texte ausgeben                                         *)
	FB_TN_SC_WRITE(	Iin_X := INT#00,
					Iin_Y := INT#03,
					Iby_ATTR := BYTE#16#70,
					Ist_STRING := 'XXXXXXXXX        MAC Address             : 00:A0:45:00:6E:9B',
					Xus_TN_SCREEN := Xus_TN_SCREEN);

	(* Statische Texte ausgeben *)
	FB_TN_SC_WRITE(	Iin_X := INT#00,
					Iin_Y := INT#04,
					Iby_ATTR := BYTE#16#70,
					Ist_STRING := 'X   X  XX',
					Xus_TN_SCREEN := Xus_TN_SCREEN);

	(* Statische Texte ausgeben *)
	FB_TN_SC_WRITE(	Iin_X := INT#00,
					Iin_Y := INT#05,
					Iby_ATTR := BYTE#16#70,
					Ist_STRING := 'X   O   X',
					Xus_TN_SCREEN := Xus_TN_SCREEN);

	(* Statische Texte ausgeben *)
	FB_TN_SC_WRITE(	Iin_X := INT#00,
					Iin_Y := INT#06,
					Iby_ATTR := BYTE#16#70,
					Ist_STRING := 'X   X  XX',
					Xus_TN_SCREEN := Xus_TN_SCREEN);

	(* Statische Texte ausgeben *)
	FB_TN_SC_WRITE(	Iin_X := INT#00,
					Iin_Y := INT#07,
					Iby_ATTR := BYTE#16#70,
					Ist_STRING := 'X   XXXXX',
					Xus_TN_SCREEN := Xus_TN_SCREEN);

	(* Statische Texte ausgeben *)
	FB_TN_SC_WRITE(	Iin_X := INT#00,
					Iin_Y := INT#08,
					Iby_ATTR := BYTE#16#70,
					Ist_STRING := 'X   XXXXX',
					Xus_TN_SCREEN := Xus_TN_SCREEN);

	(* Statische Texte ausgeben *)
	FB_TN_SC_WRITE(	Iin_X := INT#00,
					Iin_Y := INT#09,
					Iby_ATTR := BYTE#16#70,
					Ist_STRING := 'XXXXXXXXX',
					Xus_TN_SCREEN := Xus_TN_SCREEN);

	(* Alle Input-Controls initialisieren *)

	Xus_TN_INPUT_CONTROL.bo_Enable      := FALSE;

	Xus_TN_INPUT_CONTROL.usa_TN_INPUT_CONTROL_DATA[1].in_Type := INT#01;
	Xus_TN_INPUT_CONTROL.usa_TN_INPUT_CONTROL_DATA[1].in_Y := INT#04;
	Xus_TN_INPUT_CONTROL.usa_TN_INPUT_CONTROL_DATA[1].in_X := INT#44;
	Xus_TN_INPUT_CONTROL.usa_TN_INPUT_CONTROL_DATA[1].by_Attr_mF := BYTE#16#07; (* Weiss, Grün *)
	Xus_TN_INPUT_CONTROL.usa_TN_INPUT_CONTROL_DATA[1].by_Attr_oF := BYTE#16#70; (* Weiss, Blau *)
	Xus_TN_INPUT_CONTROL.usa_TN_INPUT_CONTROL_DATA[1].in_Cursor_Pos := INT#0;
	Xus_TN_INPUT_CONTROL.usa_TN_INPUT_CONTROL_DATA[1].bo_Input_Only_Num := TRUE;
	Xus_TN_INPUT_CONTROL.usa_TN_INPUT_CONTROL_DATA[1].bo_Input_Hidden := FALSE;
	Xus_TN_INPUT_CONTROL.usa_TN_INPUT_CONTROL_DATA[1].st_Input_Mask := '   .   .   .   ';
	Xus_TN_INPUT_CONTROL.usa_TN_INPUT_CONTROL_DATA[1].st_Input_Data := Xus_TN_INPUT_CONTROL.usa_TN_INPUT_CONTROL_DATA[1].st_Input_Mask;
	Xus_TN_INPUT_CONTROL.usa_TN_INPUT_CONTROL_DATA[1].st_Input_ToolTip := 'Enter Agent IP Address in decimal dot format (e.g., 209.131.209.13)';
	Xus_TN_INPUT_CONTROL.usa_TN_INPUT_CONTROL_DATA[1].in_Input_Option := INT#01;
	Xus_TN_INPUT_CONTROL.usa_TN_INPUT_CONTROL_DATA[1].in_Title_Y_Offset := INT#00;
	Xus_TN_INPUT_CONTROL.usa_TN_INPUT_CONTROL_DATA[1].in_Title_X_Offset := -27;
	Xus_TN_INPUT_CONTROL.usa_TN_INPUT_CONTROL_DATA[1].by_Title_Attr := BYTE#16#70;
	Xus_TN_INPUT_CONTROL.usa_TN_INPUT_CONTROL_DATA[1].st_Title_String := 'IP Address              : [149.208.100.100]';

	Xus_TN_INPUT_CONTROL.usa_TN_INPUT_CONTROL_DATA[2].in_Type := INT#01;
	Xus_TN_INPUT_CONTROL.usa_TN_INPUT_CONTROL_DATA[2].in_Y := INT#05;
	Xus_TN_INPUT_CONTROL.usa_TN_INPUT_CONTROL_DATA[2].in_X := INT#44;
	Xus_TN_INPUT_CONTROL.usa_TN_INPUT_CONTROL_DATA[2].by_Attr_mF := BYTE#16#07; (* Weiss, Grün *)
	Xus_TN_INPUT_CONTROL.usa_TN_INPUT_CONTROL_DATA[2].by_Attr_oF := BYTE#16#70; (* Weiss, Blau *)
	Xus_TN_INPUT_CONTROL.usa_TN_INPUT_CONTROL_DATA[2].in_Cursor_Pos := INT#0;
	Xus_TN_INPUT_CONTROL.usa_TN_INPUT_CONTROL_DATA[2].bo_Input_Only_Num := TRUE;
	Xus_TN_INPUT_CONTROL.usa_TN_INPUT_CONTROL_DATA[2].bo_Input_Hidden := FALSE;
	Xus_TN_INPUT_CONTROL.usa_TN_INPUT_CONTROL_DATA[2].st_Input_Mask := '   .   .   .   ';
	Xus_TN_INPUT_CONTROL.usa_TN_INPUT_CONTROL_DATA[2].st_Input_Data := Xus_TN_INPUT_CONTROL.usa_TN_INPUT_CONTROL_DATA[1].st_Input_Mask;
	Xus_TN_INPUT_CONTROL.usa_TN_INPUT_CONTROL_DATA[2].st_Input_ToolTip := 'Enter Agent Netmask (e.g., 255.255.255.0)';
	Xus_TN_INPUT_CONTROL.usa_TN_INPUT_CONTROL_DATA[2].in_Input_Option := INT#01;
	Xus_TN_INPUT_CONTROL.usa_TN_INPUT_CONTROL_DATA[2].in_Title_Y_Offset := INT#00;
	Xus_TN_INPUT_CONTROL.usa_TN_INPUT_CONTROL_DATA[2].in_Title_X_Offset := -27;
	Xus_TN_INPUT_CONTROL.usa_TN_INPUT_CONTROL_DATA[2].by_Title_Attr := BYTE#16#70;
	Xus_TN_INPUT_CONTROL.usa_TN_INPUT_CONTROL_DATA[2].st_Title_String := 'Subnet Mask             : [255.255.255.128]';

	Xus_TN_INPUT_CONTROL.usa_TN_INPUT_CONTROL_DATA[3].in_Type := INT#01;
	Xus_TN_INPUT_CONTROL.usa_TN_INPUT_CONTROL_DATA[3].in_Y := INT#06;
	Xus_TN_INPUT_CONTROL.usa_TN_INPUT_CONTROL_DATA[3].in_X := INT#44;
	Xus_TN_INPUT_CONTROL.usa_TN_INPUT_CONTROL_DATA[3].by_Attr_mF := BYTE#16#07; (* Weiss, Grün *)
	Xus_TN_INPUT_CONTROL.usa_TN_INPUT_CONTROL_DATA[3].by_Attr_oF := BYTE#16#70; (* Weiss, Blau *)
	Xus_TN_INPUT_CONTROL.usa_TN_INPUT_CONTROL_DATA[3].in_Cursor_Pos := INT#0;
	Xus_TN_INPUT_CONTROL.usa_TN_INPUT_CONTROL_DATA[3].bo_Input_Only_Num := TRUE;
	Xus_TN_INPUT_CONTROL.usa_TN_INPUT_CONTROL_DATA[3].bo_Input_Hidden := FALSE;
	Xus_TN_INPUT_CONTROL.usa_TN_INPUT_CONTROL_DATA[3].st_Input_Mask := '   .   .   .   ';
	Xus_TN_INPUT_CONTROL.usa_TN_INPUT_CONTROL_DATA[3].st_Input_Data := Xus_TN_INPUT_CONTROL.usa_TN_INPUT_CONTROL_DATA[1].st_Input_Mask;
	Xus_TN_INPUT_CONTROL.usa_TN_INPUT_CONTROL_DATA[3].st_Input_ToolTip := 'Enter Agent Default Gateway, (e.g., 209.131.209.1)';
	Xus_TN_INPUT_CONTROL.usa_TN_INPUT_CONTROL_DATA[3].in_Input_Option := INT#01;
	Xus_TN_INPUT_CONTROL.usa_TN_INPUT_CONTROL_DATA[3].in_Title_Y_Offset := INT#00;
	Xus_TN_INPUT_CONTROL.usa_TN_INPUT_CONTROL_DATA[3].in_Title_X_Offset := -27;
	Xus_TN_INPUT_CONTROL.usa_TN_INPUT_CONTROL_DATA[3].by_Title_Attr := BYTE#16#70;
	Xus_TN_INPUT_CONTROL.usa_TN_INPUT_CONTROL_DATA[3].st_Title_String := 'Default Gateway         : [149.208.100.1  ]';

	Xus_TN_INPUT_CONTROL.usa_TN_INPUT_CONTROL_DATA[4].in_Type := INT#02;
	Xus_TN_INPUT_CONTROL.usa_TN_INPUT_CONTROL_DATA[4].in_Y := INT#07;
	Xus_TN_INPUT_CONTROL.usa_TN_INPUT_CONTROL_DATA[4].in_X := INT#44;
	Xus_TN_INPUT_CONTROL.usa_TN_INPUT_CONTROL_DATA[4].by_Attr_mF := BYTE#16#07;
	Xus_TN_INPUT_CONTROL.usa_TN_INPUT_CONTROL_DATA[4].by_Attr_oF := BYTE#16#70;
	Xus_TN_INPUT_CONTROL.usa_TN_INPUT_CONTROL_DATA[4].st_Input_Mask := '       ';
	Xus_TN_INPUT_CONTROL.usa_TN_INPUT_CONTROL_DATA[4].st_Input_Data := 'BootP  #DHCP   #DCP    #Static ';
	Xus_TN_INPUT_CONTROL.usa_TN_INPUT_CONTROL_DATA[4].st_Input_ToolTip := 'Push SPACE to select the address assignment (effective after reboot)';
	Xus_TN_INPUT_CONTROL.usa_TN_INPUT_CONTROL_DATA[4].in_Input_Option := INT#02;
	Xus_TN_INPUT_CONTROL.usa_TN_INPUT_CONTROL_DATA[4].in_Title_Y_Offset := INT#00;
	Xus_TN_INPUT_CONTROL.usa_TN_INPUT_CONTROL_DATA[4].in_Title_X_Offset := -27;
	Xus_TN_INPUT_CONTROL.usa_TN_INPUT_CONTROL_DATA[4].by_Title_Attr := BYTE#16#70;
	Xus_TN_INPUT_CONTROL.usa_TN_INPUT_CONTROL_DATA[4].st_Title_String := 'IP Parameter Assignment : <BootP  >';

	Xus_TN_INPUT_CONTROL.usa_TN_INPUT_CONTROL_DATA[5].in_Type := INT#02;
	Xus_TN_INPUT_CONTROL.usa_TN_INPUT_CONTROL_DATA[5].in_Y := INT#09;
	Xus_TN_INPUT_CONTROL.usa_TN_INPUT_CONTROL_DATA[5].in_X := INT#44;
	Xus_TN_INPUT_CONTROL.usa_TN_INPUT_CONTROL_DATA[5].by_Attr_mF := BYTE#16#07;
	Xus_TN_INPUT_CONTROL.usa_TN_INPUT_CONTROL_DATA[5].by_Attr_oF := BYTE#16#70;
	Xus_TN_INPUT_CONTROL.usa_TN_INPUT_CONTROL_DATA[5].st_Input_Mask := '                              ';
	Xus_TN_INPUT_CONTROL.usa_TN_INPUT_CONTROL_DATA[5].st_Input_Data := 'No Redundancy#Rapid Spanning Tree, Disabled#Rapid Spanning Tree, Enabled';
	Xus_TN_INPUT_CONTROL.usa_TN_INPUT_CONTROL_DATA[5].st_Input_ToolTip := 'Push SPACE to chose redundancy (network disruption for few seconds if enabled)';
	Xus_TN_INPUT_CONTROL.usa_TN_INPUT_CONTROL_DATA[5].in_Input_Option := INT#02;
	Xus_TN_INPUT_CONTROL.usa_TN_INPUT_CONTROL_DATA[5].in_Title_Y_Offset := INT#00;
	Xus_TN_INPUT_CONTROL.usa_TN_INPUT_CONTROL_DATA[5].in_Title_X_Offset := -27;
	Xus_TN_INPUT_CONTROL.usa_TN_INPUT_CONTROL_DATA[5].by_Title_Attr := BYTE#16#70;
	Xus_TN_INPUT_CONTROL.usa_TN_INPUT_CONTROL_DATA[5].st_Title_String := 'Redundancy              : <No Redundancy                 >';

	(* Statische Texte ausgeben *)
	FB_TN_SC_WRITE(	Iin_X := INT#17,
					Iin_Y := INT#10,
					Iby_ATTR := BYTE#16#70,
					Ist_STRING := 'Current Vlan Status     :  VLAN Transparent',
					Xus_TN_SCREEN := Xus_TN_SCREEN);

	Xus_TN_INPUT_CONTROL.usa_TN_INPUT_CONTROL_DATA[6].in_Type := INT#02;
	Xus_TN_INPUT_CONTROL.usa_TN_INPUT_CONTROL_DATA[6].in_Y := INT#11;
	Xus_TN_INPUT_CONTROL.usa_TN_INPUT_CONTROL_DATA[6].in_X := INT#44;
	Xus_TN_INPUT_CONTROL.usa_TN_INPUT_CONTROL_DATA[6].by_Attr_mF := BYTE#16#07;
	Xus_TN_INPUT_CONTROL.usa_TN_INPUT_CONTROL_DATA[6].by_Attr_oF := BYTE#16#70;
	Xus_TN_INPUT_CONTROL.usa_TN_INPUT_CONTROL_DATA[6].st_Input_Mask := '                        ';
	Xus_TN_INPUT_CONTROL.usa_TN_INPUT_CONTROL_DATA[6].st_Input_Data := 'VLAN Transparent#VLAN Tagging';
	Xus_TN_INPUT_CONTROL.usa_TN_INPUT_CONTROL_DATA[6].st_Input_ToolTip := 'Push SPACE to toggle the VLAN Mode (effective after reboot)';
	Xus_TN_INPUT_CONTROL.usa_TN_INPUT_CONTROL_DATA[6].in_Input_Option := INT#02;
	Xus_TN_INPUT_CONTROL.usa_TN_INPUT_CONTROL_DATA[6].in_Title_Y_Offset := INT#00;
	Xus_TN_INPUT_CONTROL.usa_TN_INPUT_CONTROL_DATA[6].in_Title_X_Offset := -27;
	Xus_TN_INPUT_CONTROL.usa_TN_INPUT_CONTROL_DATA[6].by_Title_Attr := BYTE#16#70;
	Xus_TN_INPUT_CONTROL.usa_TN_INPUT_CONTROL_DATA[6].st_Title_String := 'Vlan Mode               : <VLAN Transparent        >';

	Xus_TN_INPUT_CONTROL.usa_TN_INPUT_CONTROL_DATA[7].in_Type := INT#02;
	Xus_TN_INPUT_CONTROL.usa_TN_INPUT_CONTROL_DATA[7].in_Y := INT#12;
	Xus_TN_INPUT_CONTROL.usa_TN_INPUT_CONTROL_DATA[7].in_X := INT#44;
	Xus_TN_INPUT_CONTROL.usa_TN_INPUT_CONTROL_DATA[7].by_Attr_mF := BYTE#16#07;
	Xus_TN_INPUT_CONTROL.usa_TN_INPUT_CONTROL_DATA[7].by_Attr_oF := BYTE#16#70;
	Xus_TN_INPUT_CONTROL.usa_TN_INPUT_CONTROL_DATA[7].st_Input_Mask := '       ';
	Xus_TN_INPUT_CONTROL.usa_TN_INPUT_CONTROL_DATA[7].st_Input_Data := 'Disable#Enable';
	Xus_TN_INPUT_CONTROL.usa_TN_INPUT_CONTROL_DATA[7].st_Input_ToolTip := 'Push SPACE to Enable/Disable Port Security';
	Xus_TN_INPUT_CONTROL.usa_TN_INPUT_CONTROL_DATA[7].in_Input_Option := INT#02;
	Xus_TN_INPUT_CONTROL.usa_TN_INPUT_CONTROL_DATA[7].in_Title_Y_Offset := INT#00;
	Xus_TN_INPUT_CONTROL.usa_TN_INPUT_CONTROL_DATA[7].in_Title_X_Offset := -27;
	Xus_TN_INPUT_CONTROL.usa_TN_INPUT_CONTROL_DATA[7].by_Title_Attr := BYTE#16#70;
	Xus_TN_INPUT_CONTROL.usa_TN_INPUT_CONTROL_DATA[7].st_Title_String := 'Port Security           : <Disable>';

	Xus_TN_INPUT_CONTROL.usa_TN_INPUT_CONTROL_DATA[8].in_Type := INT#02;
	Xus_TN_INPUT_CONTROL.usa_TN_INPUT_CONTROL_DATA[8].in_Y := INT#13;
	Xus_TN_INPUT_CONTROL.usa_TN_INPUT_CONTROL_DATA[8].in_X := INT#44;
	Xus_TN_INPUT_CONTROL.usa_TN_INPUT_CONTROL_DATA[8].by_Attr_mF := BYTE#16#07;
	Xus_TN_INPUT_CONTROL.usa_TN_INPUT_CONTROL_DATA[8].by_Attr_oF := BYTE#16#70;
	Xus_TN_INPUT_CONTROL.usa_TN_INPUT_CONTROL_DATA[8].st_Input_Mask := '       ';
	Xus_TN_INPUT_CONTROL.usa_TN_INPUT_CONTROL_DATA[8].st_Input_Data := 'Disable#Enable';
	Xus_TN_INPUT_CONTROL.usa_TN_INPUT_CONTROL_DATA[8].st_Input_ToolTip := 'Push SPACE to Enable/Disable Access Control for the WEB Interface';
	Xus_TN_INPUT_CONTROL.usa_TN_INPUT_CONTROL_DATA[8].in_Input_Option := INT#02;
	Xus_TN_INPUT_CONTROL.usa_TN_INPUT_CONTROL_DATA[8].in_Title_Y_Offset := INT#00;
	Xus_TN_INPUT_CONTROL.usa_TN_INPUT_CONTROL_DATA[8].in_Title_X_Offset := -27;
	Xus_TN_INPUT_CONTROL.usa_TN_INPUT_CONTROL_DATA[8].by_Title_Attr := BYTE#16#70;
	Xus_TN_INPUT_CONTROL.usa_TN_INPUT_CONTROL_DATA[8].st_Title_String := 'Access Control for Web  : <Disable>';

	Xus_TN_INPUT_CONTROL.usa_TN_INPUT_CONTROL_DATA[9].in_Type := INT#02;
	Xus_TN_INPUT_CONTROL.usa_TN_INPUT_CONTROL_DATA[9].in_Y := INT#14;
	Xus_TN_INPUT_CONTROL.usa_TN_INPUT_CONTROL_DATA[9].in_X := INT#44;
	Xus_TN_INPUT_CONTROL.usa_TN_INPUT_CONTROL_DATA[9].by_Attr_mF := BYTE#16#07;
	Xus_TN_INPUT_CONTROL.usa_TN_INPUT_CONTROL_DATA[9].by_Attr_oF := BYTE#16#70;
	Xus_TN_INPUT_CONTROL.usa_TN_INPUT_CONTROL_DATA[9].st_Input_Mask := '        ';
	Xus_TN_INPUT_CONTROL.usa_TN_INPUT_CONTROL_DATA[9].st_Input_Data := 'Default#Profinet';
	Xus_TN_INPUT_CONTROL.usa_TN_INPUT_CONTROL_DATA[9].st_Input_ToolTip := 'Push SPACE to select the switch operating mode';
	Xus_TN_INPUT_CONTROL.usa_TN_INPUT_CONTROL_DATA[9].in_Input_Option := INT#02;
	Xus_TN_INPUT_CONTROL.usa_TN_INPUT_CONTROL_DATA[9].in_Title_Y_Offset := INT#00;
	Xus_TN_INPUT_CONTROL.usa_TN_INPUT_CONTROL_DATA[9].in_Title_X_Offset := -27;
	Xus_TN_INPUT_CONTROL.usa_TN_INPUT_CONTROL_DATA[9].by_Title_Attr := BYTE#16#70;
	Xus_TN_INPUT_CONTROL.usa_TN_INPUT_CONTROL_DATA[9].st_Title_String := 'Switch Operating Mode   : <Default >';

	Xus_TN_INPUT_CONTROL.usa_TN_INPUT_CONTROL_DATA[10].in_Type := INT#02;
	Xus_TN_INPUT_CONTROL.usa_TN_INPUT_CONTROL_DATA[10].in_Y := INT#16;
	Xus_TN_INPUT_CONTROL.usa_TN_INPUT_CONTROL_DATA[10].in_X := INT#44;
	Xus_TN_INPUT_CONTROL.usa_TN_INPUT_CONTROL_DATA[10].by_Attr_mF := BYTE#16#07;
	Xus_TN_INPUT_CONTROL.usa_TN_INPUT_CONTROL_DATA[10].by_Attr_oF := BYTE#16#70;
	Xus_TN_INPUT_CONTROL.usa_TN_INPUT_CONTROL_DATA[10].st_Input_Mask := '       ';
	Xus_TN_INPUT_CONTROL.usa_TN_INPUT_CONTROL_DATA[10].st_Input_Data := 'Enable#Disable';
	Xus_TN_INPUT_CONTROL.usa_TN_INPUT_CONTROL_DATA[10].st_Input_ToolTip := 'Push SPACE to Enable/Disable Web Interface (effective after reboot)';
	Xus_TN_INPUT_CONTROL.usa_TN_INPUT_CONTROL_DATA[10].in_Input_Option := INT#02;
	Xus_TN_INPUT_CONTROL.usa_TN_INPUT_CONTROL_DATA[10].in_Title_Y_Offset := INT#00;
	Xus_TN_INPUT_CONTROL.usa_TN_INPUT_CONTROL_DATA[10].in_Title_X_Offset := -27;
	Xus_TN_INPUT_CONTROL.usa_TN_INPUT_CONTROL_DATA[10].by_Title_Attr := BYTE#16#70;
	Xus_TN_INPUT_CONTROL.usa_TN_INPUT_CONTROL_DATA[10].st_Title_String := 'Web Interface           : <Enable >';

	Xus_TN_INPUT_CONTROL.usa_TN_INPUT_CONTROL_DATA[11].in_Type := INT#02;
	Xus_TN_INPUT_CONTROL.usa_TN_INPUT_CONTROL_DATA[11].in_Y := INT#17;
	Xus_TN_INPUT_CONTROL.usa_TN_INPUT_CONTROL_DATA[11].in_X := INT#44;
	Xus_TN_INPUT_CONTROL.usa_TN_INPUT_CONTROL_DATA[11].by_Attr_mF := BYTE#16#07;
	Xus_TN_INPUT_CONTROL.usa_TN_INPUT_CONTROL_DATA[11].by_Attr_oF := BYTE#16#70;
	Xus_TN_INPUT_CONTROL.usa_TN_INPUT_CONTROL_DATA[11].st_Input_Mask := '       ';
	Xus_TN_INPUT_CONTROL.usa_TN_INPUT_CONTROL_DATA[11].st_Input_Data := 'Enable#Disable';
	Xus_TN_INPUT_CONTROL.usa_TN_INPUT_CONTROL_DATA[11].st_Input_ToolTip := 'Push SPACE to Enable/Disable Telnet Interface (effective after reboot)';
	Xus_TN_INPUT_CONTROL.usa_TN_INPUT_CONTROL_DATA[11].in_Input_Option := INT#02;
	Xus_TN_INPUT_CONTROL.usa_TN_INPUT_CONTROL_DATA[11].in_Title_Y_Offset := INT#00;
	Xus_TN_INPUT_CONTROL.usa_TN_INPUT_CONTROL_DATA[11].in_Title_X_Offset := -27;
	Xus_TN_INPUT_CONTROL.usa_TN_INPUT_CONTROL_DATA[11].by_Title_Attr := BYTE#16#70;
	Xus_TN_INPUT_CONTROL.usa_TN_INPUT_CONTROL_DATA[11].st_Title_String := 'Telnet Interface        : <Enable >';

	Xus_TN_INPUT_CONTROL.usa_TN_INPUT_CONTROL_DATA[12].in_Type := INT#02;
	Xus_TN_INPUT_CONTROL.usa_TN_INPUT_CONTROL_DATA[12].in_Y := INT#18;
	Xus_TN_INPUT_CONTROL.usa_TN_INPUT_CONTROL_DATA[12].in_X := INT#44;
	Xus_TN_INPUT_CONTROL.usa_TN_INPUT_CONTROL_DATA[12].by_Attr_mF := BYTE#16#07;
	Xus_TN_INPUT_CONTROL.usa_TN_INPUT_CONTROL_DATA[12].by_Attr_oF := BYTE#16#70;
	Xus_TN_INPUT_CONTROL.usa_TN_INPUT_CONTROL_DATA[12].st_Input_Mask := '       ';
	Xus_TN_INPUT_CONTROL.usa_TN_INPUT_CONTROL_DATA[12].st_Input_Data := 'Enable#Disable';
	Xus_TN_INPUT_CONTROL.usa_TN_INPUT_CONTROL_DATA[12].st_Input_ToolTip := 'Push SPACE to Enable/Disable SNMP Interface (effective after reboot)';
	Xus_TN_INPUT_CONTROL.usa_TN_INPUT_CONTROL_DATA[12].in_Input_Option := INT#02;
	Xus_TN_INPUT_CONTROL.usa_TN_INPUT_CONTROL_DATA[12].in_Title_Y_Offset := INT#00;
	Xus_TN_INPUT_CONTROL.usa_TN_INPUT_CONTROL_DATA[12].in_Title_X_Offset := -27;
	Xus_TN_INPUT_CONTROL.usa_TN_INPUT_CONTROL_DATA[12].by_Title_Attr := BYTE#16#70;
	Xus_TN_INPUT_CONTROL.usa_TN_INPUT_CONTROL_DATA[12].st_Title_String := 'SNMP Interface          : <Enable >';

	Xus_TN_INPUT_CONTROL.usa_TN_INPUT_CONTROL_DATA[13].in_Type := INT#02;
	Xus_TN_INPUT_CONTROL.usa_TN_INPUT_CONTROL_DATA[13].in_Y := INT#20;
	Xus_TN_INPUT_CONTROL.usa_TN_INPUT_CONTROL_DATA[13].in_X := INT#44;
	Xus_TN_INPUT_CONTROL.usa_TN_INPUT_CONTROL_DATA[13].by_Attr_mF := BYTE#16#07;
	Xus_TN_INPUT_CONTROL.usa_TN_INPUT_CONTROL_DATA[13].by_Attr_oF := BYTE#16#70;
	Xus_TN_INPUT_CONTROL.usa_TN_INPUT_CONTROL_DATA[13].st_Input_Mask := '                                 ';
	Xus_TN_INPUT_CONTROL.usa_TN_INPUT_CONTROL_DATA[13].st_Input_Data := 'No reset#Reset Switch#Reset Switch to factory defaults';
	Xus_TN_INPUT_CONTROL.usa_TN_INPUT_CONTROL_DATA[13].st_Input_ToolTip := 'Push SPACE to select Reset Option';
	Xus_TN_INPUT_CONTROL.usa_TN_INPUT_CONTROL_DATA[13].in_Input_Option := INT#02;
	Xus_TN_INPUT_CONTROL.usa_TN_INPUT_CONTROL_DATA[13].in_Title_Y_Offset := INT#00;
	Xus_TN_INPUT_CONTROL.usa_TN_INPUT_CONTROL_DATA[13].in_Title_X_Offset := -27;
	Xus_TN_INPUT_CONTROL.usa_TN_INPUT_CONTROL_DATA[13].by_Title_Attr := BYTE#16#70;
	Xus_TN_INPUT_CONTROL.usa_TN_INPUT_CONTROL_DATA[13].st_Title_String := 'Reset                   : <No reset                         >';

	Xus_TN_INPUT_CONTROL.usa_TN_INPUT_CONTROL_DATA[14].in_Type := INT#02;
	Xus_TN_INPUT_CONTROL.usa_TN_INPUT_CONTROL_DATA[14].in_Y := INT#22;
	Xus_TN_INPUT_CONTROL.usa_TN_INPUT_CONTROL_DATA[14].in_X := INT#18;
	Xus_TN_INPUT_CONTROL.usa_TN_INPUT_CONTROL_DATA[14].by_Attr_mF := BYTE#16#07;
	Xus_TN_INPUT_CONTROL.usa_TN_INPUT_CONTROL_DATA[14].by_Attr_oF := BYTE#16#70;
	Xus_TN_INPUT_CONTROL.usa_TN_INPUT_CONTROL_DATA[14].st_Input_ToolTip := 'Apply and save ALL changes to permanent memory';
	Xus_TN_INPUT_CONTROL.usa_TN_INPUT_CONTROL_DATA[14].in_Input_Option := INT#01;
	Xus_TN_INPUT_CONTROL.usa_TN_INPUT_CONTROL_DATA[14].in_Title_Y_Offset := INT#00;
	Xus_TN_INPUT_CONTROL.usa_TN_INPUT_CONTROL_DATA[14].in_Title_X_Offset := INT#00;
	Xus_TN_INPUT_CONTROL.usa_TN_INPUT_CONTROL_DATA[14].by_Title_Attr := BYTE#16#70;
	Xus_TN_INPUT_CONTROL.usa_TN_INPUT_CONTROL_DATA[14].st_Title_String := '';
	Xus_TN_INPUT_CONTROL.usa_TN_INPUT_CONTROL_DATA[14].st_Input_Mask := '    ';
	Xus_TN_INPUT_CONTROL.usa_TN_INPUT_CONTROL_DATA[14].st_Input_Data := 'SAVE';

	Xus_TN_INPUT_CONTROL.usa_TN_INPUT_CONTROL_DATA[15].in_Type := INT#02;
	Xus_TN_INPUT_CONTROL.usa_TN_INPUT_CONTROL_DATA[15].in_Y := INT#22;
	Xus_TN_INPUT_CONTROL.usa_TN_INPUT_CONTROL_DATA[15].in_X := INT#11;
	Xus_TN_INPUT_CONTROL.usa_TN_INPUT_CONTROL_DATA[15].by_Attr_mF := BYTE#16#07;
	Xus_TN_INPUT_CONTROL.usa_TN_INPUT_CONTROL_DATA[15].by_Attr_oF := BYTE#16#70;
	Xus_TN_INPUT_CONTROL.usa_TN_INPUT_CONTROL_DATA[15].st_Input_ToolTip := 'Apply changes';
	Xus_TN_INPUT_CONTROL.usa_TN_INPUT_CONTROL_DATA[15].in_Input_Option := INT#01;
	Xus_TN_INPUT_CONTROL.usa_TN_INPUT_CONTROL_DATA[15].in_Title_Y_Offset := INT#00;
	Xus_TN_INPUT_CONTROL.usa_TN_INPUT_CONTROL_DATA[15].in_Title_X_Offset := INT#00;
	Xus_TN_INPUT_CONTROL.usa_TN_INPUT_CONTROL_DATA[15].by_Title_Attr := BYTE#16#70;
	Xus_TN_INPUT_CONTROL.usa_TN_INPUT_CONTROL_DATA[15].st_Title_String := '';
	Xus_TN_INPUT_CONTROL.usa_TN_INPUT_CONTROL_DATA[15].st_Input_Mask := '     ';
	Xus_TN_INPUT_CONTROL.usa_TN_INPUT_CONTROL_DATA[15].st_Input_Data := 'APPLY';

	Xus_TN_INPUT_CONTROL.usa_TN_INPUT_CONTROL_DATA[16].in_Type := INT#02;
	Xus_TN_INPUT_CONTROL.usa_TN_INPUT_CONTROL_DATA[16].in_Y := INT#22;
	Xus_TN_INPUT_CONTROL.usa_TN_INPUT_CONTROL_DATA[16].in_X := INT#03;
	Xus_TN_INPUT_CONTROL.usa_TN_INPUT_CONTROL_DATA[16].by_Attr_mF := BYTE#16#07;
	Xus_TN_INPUT_CONTROL.usa_TN_INPUT_CONTROL_DATA[16].by_Attr_oF := BYTE#16#70;
	Xus_TN_INPUT_CONTROL.usa_TN_INPUT_CONTROL_DATA[16].st_Input_ToolTip := 'Return to Main Menu';
	Xus_TN_INPUT_CONTROL.usa_TN_INPUT_CONTROL_DATA[16].in_Input_Option := INT#01;
	Xus_TN_INPUT_CONTROL.usa_TN_INPUT_CONTROL_DATA[16].in_Title_Y_Offset := INT#00;
	Xus_TN_INPUT_CONTROL.usa_TN_INPUT_CONTROL_DATA[16].in_Title_X_Offset := INT#00;
	Xus_TN_INPUT_CONTROL.usa_TN_INPUT_CONTROL_DATA[16].by_Title_Attr := BYTE#16#70;
	Xus_TN_INPUT_CONTROL.usa_TN_INPUT_CONTROL_DATA[16].st_Title_String := '';
	Xus_TN_INPUT_CONTROL.usa_TN_INPUT_CONTROL_DATA[16].st_Input_Mask := '      ';
	Xus_TN_INPUT_CONTROL.usa_TN_INPUT_CONTROL_DATA[16].st_Input_Data := 'LOGOUT';

	(* Control-Tool-Tip *)
	Xus_TN_INPUT_CONTROL.in_ToolTip_Y := INT#23;
	Xus_TN_INPUT_CONTROL.in_ToolTip_X := INT#00;
	Xus_TN_INPUT_CONTROL.by_ToolTip_Attr := BYTE#07;
	Xus_TN_INPUT_CONTROL.in_ToolTip_Size := INT#80;

	(* Control-Verwaltung initialisieren *)
	Xus_TN_INPUT_CONTROL.in_Count := INT#16;
	Xus_TN_INPUT_CONTROL.bo_Enable := TRUE;
	Xus_TN_INPUT_CONTROL.bo_Reset_Fokus := TRUE;

END_IF;

IF (Xus_TN_SCREEN.in_Page_Number = INT#05) THEN

	(* eingegebenen String übernehmen *)
	IF Xus_TN_INPUT_CONTROL.usa_TN_INPUT_CONTROL_DATA[16].bo_Input_Entered = TRUE THEN

		Xus_TN_INPUT_CONTROL.usa_TN_INPUT_CONTROL_DATA[16].bo_Input_Entered := FALSE;
		Xus_TN_SCREEN.in_Page_Number := INT#00;
	END_IF;
END_IF;
END_PROGRAM

(* POU WORLD_WEATHER_DEMO, CFC *)
PROGRAM WORLD_WEATHER_DEMO
VAR
	IP_C: IP_C;
	S_BUF: NETWORK_BUFFER;
	R_BUF: NETWORK_BUFFER;
	IP_CONTROL_1: IP_CONTROL;
	TON_1: TON;
	activate: BOOL := TRUE;
	COUNT_DR_1: COUNT_DR;
	done: BOOL;
	count_cycles: DWORD;
	busy: BOOL;
	error_c: DWORD;
	error_t: BYTE;
	WORLD_WEATHER: WORLD_WEATHER;
	WW_DATA: WORLD_WEATHER_DATA;
	latitude: REAL := 48.21;
	longitude: REAL := 16.37;
END_VAR
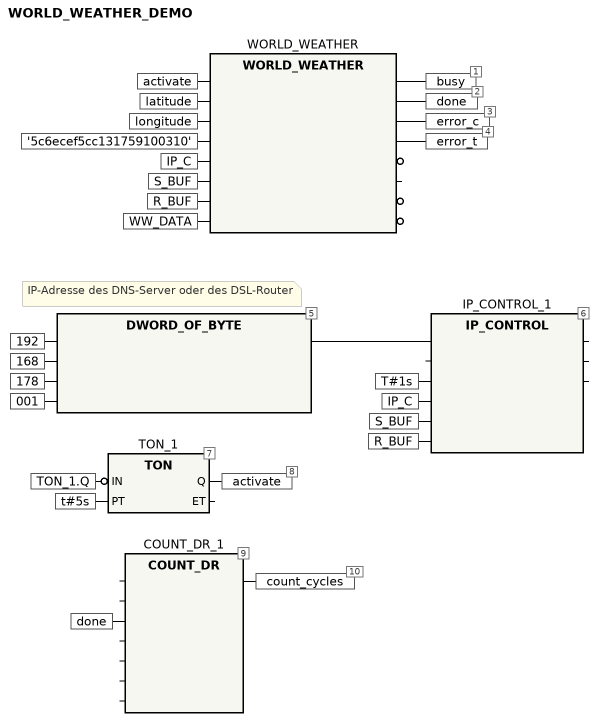
_CFC_ (* Continuous Function Chart, elements in execution order *)
(* IP-Adresse des DNS-Server oder des DSL-Router *)
#0 WORLD_WEATHER:WORLD_WEATHER(activate, latitude, longitude, '5c6ecef5cc131759100310', IP_C, S_BUF, R_BUF, WW_DATA)
#1 busy <= #0.out 1
#2 done <= #0.out 2
#3 error_c <= #0.out 3
#4 error_t <= #0.out 4
#5 DWORD_OF_BYTE(192, 168, 178, 001)
#6 IP_CONTROL_1:IP_CONTROL(#5, -, T#1s, IP_C, S_BUF, R_BUF)
#7 TON_1:TON(IN: NOT TON_1.Q, PT: t#5s)
#8 activate <= #7.Q
#9 COUNT_DR_1:COUNT_DR(-, -, done, -, -, -, -)
#10 count_cycles <= #9
_END_CFC_
END_PROGRAM

(* POU WORLD_WEATHER, ST *)
FUNCTION_BLOCK WORLD_WEATHER
VAR_IN_OUT
	IP_C : IP_C; (* IP_Control Verwaltungsstruktur *)
	S_BUF : NETWORK_BUFFER;
	R_BUF : NETWORK_BUFFER;
	WW : WORLD_WEATHER_DATA;
END_VAR
VAR_INPUT
	ACTIVATE : BOOL;
	LATITUDE : REAL;
	LONGITUDE : REAL;
	KEY : STRING(30);
END_VAR
VAR_OUTPUT
	BUSY : BOOL;
	DONE : BOOL;
	ERROR_C : DWORD;
	ERROR_T : BYTE;
END_VAR
VAR
	URL_DATA : url;
	DNS_CLIENT : DNS_CLIENT;
	HTTP_GET : HTTP_GET;
	CPB : CSV_PARSER_BUF;
	last_state : BOOL;
	value_int : INT;
	value_real : REAL;
	v_real : REAL;
	state : INT;
	url_str : STRING(STRING_LENGTH);
	offset : UDINT;
	size : INT;
	sep : BYTE;
	cnt : INT;
	day : INT;
	idx : INT;
	run : BYTE;
	result : BYTE;
	value : STRING(STRING_LENGTH);
END_VAR

(*

version 1.2		07. may 2011
programmer 		ks
tested by			ks

WORLD_WEATHER lädt von worldweather.com eine Wetter csv-datei und analysiert die Daten und legt diese in einem Array ab
Die Wetterdaten werden für 5 tage aufbereitet
*)
CASE state OF

00:
	IF ACTIVATE AND NOT last_state THEN
		state := 20;
		DONE := FALSE;
		BUSY := TRUE;
		ERROR_C := DWORD#0;
		ERROR_T := BYTE#0;
	END_IF;

20: (* URL for DNS UND HTTP-GET *)
	(* Example: http://free.worldweatheronline.com/feed/weather.ashx?q=48.21,16.37&format=csv&num_of_days=5&key=xxxxxxxxxxxxxxxxxxxxxx *)
	url_str := CONCAT('http://free.worldweatheronline.com/feed/weather.ashx?q=',REAL_TO_STRF(LATITUDE,6));
	url_str := CONCAT(url_str,',');
	url_str := CONCAT(url_str,REAL_TO_STRF(LONGITUDE,6));
	url_str := CONCAT(url_str,'&format=csv&num_of_days=5&key=');
	url_str := CONCAT(url_str,key);

	URL_DATA:=STRING_TO_URL(STR:=url_str, DEFAULT_PROTOCOL:='', DEFAULT_PATH:='' );
	state := 40;

40:
	IF DNS_CLIENT.DONE THEN
		state := 60;
	ELSIF (DNS_CLIENT.ERROR > DWORD#00) THEN
		(* Fehlerbehandlung *)
		ERROR_C := DNS_CLIENT.ERROR;
	ERROR_T := BYTE#01;
		state   := 100;
	END_IF;

60:
	IF HTTP_GET.DONE THEN
		sep := 0;
		idx := 0;
		day := 0;
		cnt := 0;
		OFFSET := HTTP_GET.BODY_START; (* Start Offset vorgeben *)
		size := HTTP_GET.BODY_STOP; (* End Position *)
		run := 1; (* Element suchen *)
		state := 80;

	ELSIF (HTTP_GET.ERROR > DWORD#00) THEN
		(* Fehlerbehandlung *)
		ERROR_C := HTTP_GET.ERROR;
		ERROR_T := BYTE#02;
		state := 100;
	END_IF;

80:	IF run = 0 THEN (* kein Befehl mehr aktiv ? *)
		run := 1; (*  nächstes Element suchen  *)
		IF result = 1 OR result = 2 THEN
			value_int := 0;
			value_real := 0.0;
			(* automatische konvertierung in real und int ausführen *)
			IF LEN(value) <= 20 THEN
				v_real:=FLOAT_TO_REAL(FLT:=value);
				IF CHK_REAL(v_real) = 0 THEN (* !!! prüft auf gültigen REAL Wert, ansonsten stürzt Twincat ab !!!!  *)
					value_real := v_real;
					value_int := REAL_TO_INT(value_real);
				END_IF;
			END_IF;
			cnt := cnt + 1;
			IF cnt >=8 AND cnt <= 87 THEN
				IF cnt > 22 THEN
					CASE idx OF
					00:	WW.DAY[day].DATE_OF_DAY := value;
					01:	WW.DAY[day].TEMP_MAX_C := value_int;
					02:	WW.DAY[day].TEMP_MAX_F := value_int;
					03:	WW.DAY[day].TEMP_MIN_C := value_int;
					04:	WW.DAY[day].TEMP_MIN_F := value_int;
					05:	WW.DAY[day].WIND_SPEED_MILES := value_int;
					06:	WW.DAY[day].WIND_SPEED_KMPH := value_int;
					07:	WW.DAY[day].WIND_DIR_DEGREE := value_int;
					08:	WW.DAY[day].WIND_DIR16POINT := value;
					09:	WW.DAY[day].WEATHER_CODE := value_int;
					10:	; (* weatherIconUrl auslassen *)
					11:	WW.DAY[day].WEATHER_DESC := value;
					12:	WW.DAY[day].PRECIPMM := value_real;
					END_CASE;
					idx := idx + 1;
					IF idx > 12 THEN
						idx := 0;
						day := day + 1;
					END_IF;
				ELSE
					CASE cnt OF
					08:	sep :=44; (* ab jetzt mit Trennzeichen arbeiten, *)
					09:	WW.CUR.OBSERVATION_TIME := value;
					10:	WW.CUR.TEMP_C := value_int;
					11:	WW.CUR.WEATHER_CODE := value_int;
					12:	; (* weatherIconUrl auslassen *)
					13:	WW.CUR.WEATHER_DESC := value;
					14:	WW.CUR.WIND_SPEED_MILES := value_int;
					15:	WW.CUR.WIND_SPEED_KMPH := value_int;
					16:	WW.CUR.WIND_DIR_DEGREE := value_int;
					17:	WW.CUR.WIND_DIR16POINT := value;
					18:	WW.CUR.PRECIPMM := value_real;
					19:	WW.CUR.HUMIDITY := value_int;
					20:	WW.CUR.VISIBILITY := value_int;
					21:	WW.CUR.PRESSURE := value_int;
					22:	WW.CUR.CLOUDOVER := value_int;
					END_CASE;
				END_IF;
			END_IF;
		ELSIF result = 10 THEN (* nichts mehr gefunden *)
			DONE  := TRUE;
			run := 0; (* Auswertung beenden *)
			state := 100;
		END_IF;
	END_IF;

100:
	(* UNLOCK HTTP DATA *)
	IF (NOT HTTP_GET.DONE) THEN
		state := 0;
		BUSY := FALSE;
		DONE := ERROR_T = BYTE#0;
	END_IF;

END_CASE;

(* ---------------- DNS --------------- *)
DNS_CLIENT(	IP_C:=IP_C,
			S_BUF:=S_BUF,
			R_BUF:=R_BUF,
			DOMAIN:=URL_DATA.DOMAIN,
			IP4_DNS:=DWORD#00,
			ACTIVATE:=state=40 (* DNS Start *)
			);
(* nicht oder nicht direkt verwendete Parameter *)
(*	DWORD :=DNS_CLIENT.IP4;
	BOOL  :=DNS_CLIENT.DONE;
	BYTE  :=DNS_CLIENT.ERROR; *)
(* -------------------------------------*)

(* ------------- HTTP_GET --------------- *)
HTTP_GET(	IP_C:=IP_C,
			S_BUF:=S_BUF,
			R_BUF:=R_BUF,
			IP4:=DNS_CLIENT.IP4,
			GET:=state=60,
			MODE:=BYTE#2, (* HTTP 1.1 mit persistenter Verbindung *)
			UNLOCK_BUF:=state=100,
			URL_DATA:=URL_DATA
			);

(* nicht oder nicht direkt verwendete Parameter *)
(*	STRING := HTTP_GET.HTTP_STATUS;
	UINT :=HTTP_GET.HEADER_START;
	UINT :=HTTP_GET.HEADER_STOP;
	UINT :=HTTP_GET.BODY_START;
	UINT :=HTTP_GET.BODY_STOP;
	BOOL :=HTTP_GET.DONE;
	BYTE :=HTTP_GET.ERROR;
*)
(* -------------------------------------*)
CPB(SEP:=sep,RUN:=run,OFFSET:=OFFSET,VALUE:=value,PT:=R_BUF,RESULT=>result); (* CSV PARAMETER BUF *)

last_state := ACTIVATE;

(* revision history
ks	01.oct. 2010	rev 1.0
	original version

ks	01.feb. 2011	rev 1.1
	rücksetzen von cnt 

ks	07.may. 2011	rev 1.2
	neue Domain "free.worldweatheronline.com" (Ab 30.04.2011 notwendig)
*)
END_FUNCTION_BLOCK

(* POU YAHOO_WEATHER_DEMO, CFC *)
PROGRAM YAHOO_WEATHER_DEMO
VAR
	IP_C: IP_C;
	S_BUF: NETWORK_BUFFER;
	R_BUF: NETWORK_BUFFER;
	IP_CONTROL_1: IP_CONTROL;
	TON_1: TON;
	activate: BOOL := TRUE;
	COUNT_DR_1: COUNT_DR;
	done: BOOL;
	count_cycles: DWORD;
	busy: BOOL;
	error_c: DWORD;
	error_t: BYTE;
	YAHOO_WEATHER: YAHOO_WEATHER;
	YW_DATA: YAHOO_WEATHER_DATA;
END_VAR
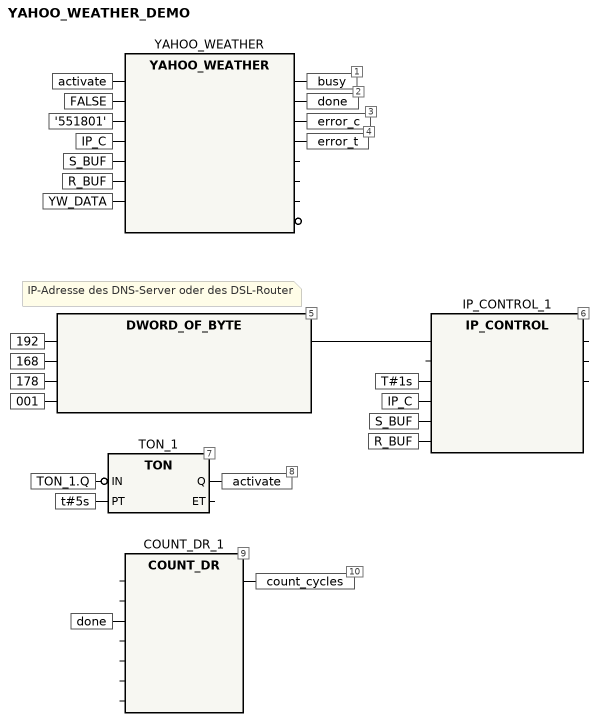
_CFC_ (* Continuous Function Chart, elements in execution order *)
(* IP-Adresse des DNS-Server oder des DSL-Router *)
#0 YAHOO_WEATHER:YAHOO_WEATHER(activate, FALSE, '551801', IP_C, S_BUF, R_BUF, YW_DATA)
#1 busy <= #0.out 1
#2 done <= #0.out 2
#3 error_c <= #0.out 3
#4 error_t <= #0.out 4
#5 DWORD_OF_BYTE(192, 168, 178, 001)
#6 IP_CONTROL_1:IP_CONTROL(#5, -, T#1s, IP_C, S_BUF, R_BUF)
#7 TON_1:TON(IN: NOT TON_1.Q, PT: t#5s)
#8 activate <= #7.Q
#9 COUNT_DR_1:COUNT_DR(-, -, done, -, -, -, -)
#10 count_cycles <= #9
_END_CFC_
END_PROGRAM

(* POU YAHOO_WEATHER, ST *)
FUNCTION_BLOCK YAHOO_WEATHER
VAR_IN_OUT
	IP_C : IP_C; (* IP_Control Verwaltungsstruktur *)
	S_BUF : NETWORK_BUFFER;
	R_BUF : NETWORK_BUFFER;
	YW : YAHOO_WEATHER_DATA;
END_VAR
VAR_INPUT
	ACTIVATE : BOOL;
	UNITS : BOOL;
	LOCATION : STRING(20);
END_VAR
VAR_OUTPUT
	BUSY : BOOL;
	DONE : BOOL;
	ERROR_C : DWORD;
	ERROR_T : BYTE;
END_VAR
VAR
	CTRL : XML_CONTROL;
	XML_READER : XML_READER;
	URL_DATA : url;
	DNS_CLIENT : DNS_CLIENT;
	HTTP_GET : HTTP_GET;
	last_state : BOOL;
	value_int : INT;
	value_real : REAL;
	v_real : REAL;
	state : INT;
END_VAR

(*

version 1.2		24. sep. 2010
programmer 		ks
tested by			ks

YAHOO_WEATHER lädt vom Yahoo-Webserver einen Wetter RSS-Feed und analysiert die Daten und legt diese in einem Array ab
*)
CASE state OF

00:	IF ACTIVATE AND NOT last_state THEN
		state := 20;
		DONE := FALSE;
		BUSY := TRUE;
		ERROR_C := DWORD#0;
		ERROR_T := BYTE#0;
	END_IF;

20: (* URL for DNS UND HTTP-GET *)
	(* Example: http://weather.yahooapis.com/forecastrss?p=94089&u=c *)
	URL_DATA:=STRING_TO_URL(STR:='http://weather.yahooapis.com/forecastrss',
							DEFAULT_PROTOCOL:='',
							DEFAULT_PATH:=''
							);
  	URL_DATA.QUERY := CONCAT('w=',LOCATION);

	IF UNITS THEN
		URL_DATA.QUERY := CONCAT(URL_DATA.QUERY,'&u=f'); (* fahrenheit *)
	ELSE
		URL_DATA.QUERY := CONCAT(URL_DATA.QUERY,'&u=c'); (* celsius *)
	END_IF;
	state := 40;

40:	IF DNS_CLIENT.DONE THEN
		state := 60;
	ELSIF (DNS_CLIENT.ERROR > DWORD#00) THEN
		(* Fehlerbehandlung *)
		ERROR_C := DNS_CLIENT.ERROR;
	ERROR_T := BYTE#01;
		state   := 100;
	END_IF;

60:	IF HTTP_GET.DONE THEN
		state := 80;
		CTRL.START_POS := HTTP_GET.BODY_START;
		CTRL.STOP_POS := HTTP_GET.BODY_STOP;
		CTRL.COMMAND := WORD#2#10000000_00011000; (* ONLY TEXT AND ATTRIBUTE *)
		CTRL.WATCHDOG  := T#1ms;

	ELSIF (HTTP_GET.ERROR > DWORD#00) THEN
		(* Fehlerbehandlung *)
		ERROR_C := HTTP_GET.ERROR;
		ERROR_T := BYTE#02;
		state := 100;
	END_IF;

80: XML_READER(CTRL:=CTRL,BUF:=R_BUF.BUFFER); (* XML Daten seriell lesen *)
	IF CTRL.TYP < 98 THEN (* nur auswerten wenn kein Watchdog durchlauf *)
		value_int := 0;
		value_real := 0.0;
		(* automatische konvertierung in real und int ausführen *)
		IF LEN(CTRL.VALUE) <= 20 THEN
			v_real:=FLOAT_TO_REAL(FLT:=CTRL.VALUE);
			IF CHK_REAL(v_real) = 0 THEN (* !!! prüft auf gültigen REAL Wert, ansonsten stürzt Twincat ab !!!!  *)
				value_real := v_real;
				value_int := REAL_TO_INT(value_real);
			END_IF;
		END_IF;

		IF CTRL.COUNT < UINT#52 THEN (* Performance-Teilung *)
			(* ------------ Teil 1 --------------*)
			CASE UINT_TO_INT(CTRL.COUNT) OF
			027: YW.TimeToLive := value_int;
			030: YW.location_city := CTRL.VALUE;
			031: YW.location_region := CTRL.VALUE;
			032: YW.location_country := CTRL.VALUE;
			035: YW.unit_temperature := CTRL.VALUE;
			036: YW.unit_distance := CTRL.VALUE;
			037: YW.unit_pressure := CTRL.VALUE;
			038: YW.unit_speed := CTRL.VALUE;
			041: YW.wind_chill := value_int;
			042: YW.wind_direction := value_int;
			043: YW.wind_speed := value_real;
			046: YW.atmosphere_humidity := value_int;
			047: YW.atmosphere_visibility := value_real;
			048: YW.atmosphere_pressure := value_int;
			049: YW.atmosphere_rising := value_int;
			END_CASE;
		ELSE
			(* ------------ Teil 2 --------------*)
			CASE UINT_TO_INT(CTRL.COUNT) OF
			052: YW.astronomy_sunrise := CTRL.VALUE;
			053: YW.astronomy_sunset := CTRL.VALUE;
			077: YW.geo_latitude := value_real;
			080: YW.geo_longitude := value_real;
			089: YW.cur_conditions_text := CTRL.VALUE; 
			090: YW.cur_conditions_code := value_int;
			091: YW.cur_conditions_temp := value_int; 
			100: YW.forcast_today_low_temp := value_int;
			101: YW.forcast_today_high_temp := value_int; 
			102: YW.forcast_today_text := CTRL.VALUE; 
			103: YW.forcast_today_code := value_int; 
			108: YW.forcast_tomorrow_low_temp := value_int; 
			109: YW.forcast_tomorrow_high_temp := value_int; 
			110: YW.forcast_tomorrow_text := CTRL.VALUE; 
			111: YW.forcast_tomorrow_code := value_int; 
			END_CASE;
		END_IF; 
	ELSIF CTRL.TYP = 99 THEN (* EXIT - letztes Element gelesen *)
		DONE  := TRUE;
		state := 100;
	END_IF; 

100:
	(* UNLOCK HTTP DATA *)
	IF (NOT HTTP_GET.DONE) THEN
		state := 0;
		BUSY := FALSE;
		DONE := ERROR_T = BYTE#0;
	END_IF; 

	END_CASE;

(* ---------------- DNS --------------- *)
DNS_CLIENT(	IP_C:=IP_C,
			S_BUF:=S_BUF,
			R_BUF:=R_BUF,
			DOMAIN:=URL_DATA.DOMAIN,
			IP4_DNS:=DWORD#00,
			ACTIVATE:=state=40 (* DNS Start *)
			);
(* nicht oder nicht direkt verwendete Parameter *)
(*	DWORD :=DNS_CLIENT.IP4;
	BOOL  :=DNS_CLIENT.DONE;
	BYTE  :=DNS_CLIENT.ERROR; *)
(* -------------------------------------*)

(* ------------- HTTP_GET --------------- *)
HTTP_GET(	IP_C:=IP_C,
			S_BUF:=S_BUF,
			R_BUF:=R_BUF,
			IP4:=DNS_CLIENT.IP4,
			GET:=state=60,
			MODE:=BYTE#2, (* HTTP 1.1 mit persistenter Verbindung *)
			UNLOCK_BUF:=state=100,
			URL_DATA:=URL_DATA
			);

(* nicht oder nicht direkt verwendete Parameter *)
(*	STRING := HTTP_GET.HTTP_STATUS;
	UINT :=HTTP_GET.HEADER_START;
	UINT :=HTTP_GET.HEADER_STOP;
	UINT :=HTTP_GET.BODY_START;
	UINT :=HTTP_GET.BODY_STOP;
	BOOL :=HTTP_GET.DONE;
	BYTE :=HTTP_GET.ERROR;
*)
(* -------------------------------------*)

last_state := ACTIVATE;

(* revision history
ks	18. dez. 2008	rev 1.0
	original version

ks	01. oct. 2009	rev 1.1
	YAHOO_WEATHER_DATA

ks	24. sep. 2010	rev 1.2
	new URL-Location-parameter and REAL_CHECK (TwinCat BUG) 
*)
END_FUNCTION_BLOCK

(* POU DLOG_STRING, ST *)
FUNCTION_BLOCK DLOG_STRING
VAR_IN_OUT
	X : DLOG_DATA;
END_VAR
VAR_INPUT
	STR : STRING;
	COLUMN : STRING;
END_VAR
VAR_OUTPUT
END_VAR
VAR
	UCB : UNI_CIRCULAR_BUFFER;
	init : BOOL;
	id : WORD;
END_VAR

(*
version 1.0		01. jan. 2011
programmer		ks
tested by			ks

DLOG_STRING legt den STRING im FIFO-RING-Buffer ab um diesen mit den Baustein DLOG_STORE_*  aufzuzeichnen
*)
IF NOT init THEN
	init := TRUE;
	X.ID_MAX := X.ID_MAX + 1;
	id := SHL(USINT_TO_WORD(X.ID_MAX),8) OR 1;
END_IF;

IF X.ADD_HEADER THEN
	X.UCB.D_STRING := COLUMN;
ELSIF X.ADD_DATA THEN
	X.UCB.D_STRING := STR;
ELSE
	RETURN;
END_IF;
X.UCB.D_HEAD := id;
X.UCB.D_MODE := 1;
UCB(DATA:=X.UCB); (* Daten eintragen *)

(* revision history
ks	01. jan. 2011	rev 1.0
	original version
*)
END_FUNCTION_BLOCK

(* POU HTML_DECODE, ST *)
FUNCTION HTML_DECODE : STRING(STRING_LENGTH)
VAR_INPUT
	IN : STRING(STRING_LENGTH);
END_VAR
VAR
	pos : INT;
	end : INT;
	tmp : STRING(10);
	code : STRING(1);
END_VAR

(*
version 1.3		10. may 2010
programmer 	hugo
tested by		oscat

HTML_DECODE converts HTML coded characters to text. 
&amp; is replaced by & ("Ampersand")
&lt; is replaced by < ("lower than")
&gt; is replaced by > ("greater than")
&quot; is replaced by " ("Quote")
all other &names characters are replaced by their respective character codes.

*)
HTML_DECODE := IN;

(* docode characters encoded by character position *)
pos := FIND(HTML_DECODE, '&');
WHILE pos > 0 DO
	tmp := MID(HTML_DECODE, 2, pos + 1);
	IF tmp = '#x' OR tmp = '#X' THEN
		(* hexadecimal representation found *)
		tmp := MID(HTML_DECODE, 10, pos + 3);
		end := FIND(tmp, ';');
		CODE := CHR_TO_STRING(DWORD_TO_BYTE(HEX_TO_DWORD(LEFT(tmp, end - 1))));
		HTML_DECODE := REPLACE(HTML_DECODE, CODE, end + 3, pos);
	ELSIF LEFT(tmp,1) = '#' THEN
		tmp := MID(HTML_DECODE, 10, pos + 2);
		end := FIND(tmp, ';');
		CODE := CHR_TO_STRING(INT_TO_BYTE(STRING_TO_INT(LEFT(tmp, end - 1))));
		HTML_DECODE := REPLACE(HTML_DECODE, CODE, end + 2, pos);
	ELSE
		(* replace all named characters *)
		tmp := MID(HTML_DECODE, 10, pos + 1);
		end := FIND(tmp, ';');
		CODE := CHR_TO_STRING(CHARCODE(LEFT(tmp, end - 1)));
		HTML_DECODE := REPLACE(HTML_DECODE, CODE, end + 1, pos);
	END_IF;
	(* search for next occurence of encoded characters *)
	pos := FINDP(HTML_DECODE, '&', pos + 1);
END_WHILE;



(* revision history
hm	3. mai. 2008	rev 1.0
	original version

hm	16. jun. 2008	rev 1.1
	changed nested call of replace for better compatibility

hm	17. dec. 2008	rev 1.2
	changed function CHR to CHR_TO_STRING

hm	10. may. 2010	rev 1.3
	stringlength 250

*)
END_FUNCTION

(* POU HTML_ENCODE, ST *)
FUNCTION HTML_ENCODE : STRING(STRING_LENGTH)
VAR_INPUT
	IN : STRING(STRING_LENGTH);
	M : BOOL;
END_VAR
VAR
	pt_in : POINTER TO ARRAY[1..255] OF BYTE;
	pt_out : POINTER TO ARRAY[1..256] OF BYTE;
	pos_in : INT;
	pos_out : INT;
	stop : INT;
	B: BYTE;
	tmp : STRING(10);
	i: INT;
END_VAR


(*
version 1.1		10. may. 2010
programmer 	hugo
tested by		hugo 

HTML_ENCODE checks a string if it contains reserved HTML characters and converts them to alternative html coding.
& is replaced by &amp; ("Ampersand")
< is replaced by &lt; ("lower than")
> is replaced by &gt; ("greater than")
" is replaced by &quot; ("Quote")

*)
pt_in  := ADR(in);
pt_out := ADR(HTML_ENCODE);

(* scan the input string and convert unallowed characters *)
pos_in := 1;
stop := LEN(in);
FOR pos_out := 1 TO 250 DO
	IF pos_in > stop THEN EXIT; END_IF;
	B := pt_in^[pos_in];
	CASE BYTE_TO_INT(B) OF
		34: (* " detected *)
			IF pos_out > STRING_LENGTH - 6 THEN EXIT; END_IF;
			pt_out^[pos_out] := 38;
			pos_out := pos_out + 1;
			pt_out^[pos_out] := 113;
			pos_out := pos_out + 1;
			pt_out^[pos_out] := 117;
			pos_out := pos_out + 1;
			pt_out^[pos_out] := 111;
			pos_out := pos_out + 1;
			pt_out^[pos_out] := 116;
			pos_out := pos_out + 1;
			pt_out^[pos_out] := 59;
		38: (* & detected *)
			IF pos_out > STRING_LENGTH - 5 THEN EXIT; END_IF;
			pt_out^[pos_out] := 38;
			pos_out := pos_out + 1;
			pt_out^[pos_out] := 97;
			pos_out := pos_out + 1;
			pt_out^[pos_out] := 109;
			pos_out := pos_out + 1;
			pt_out^[pos_out] := 112;
			pos_out := pos_out + 1;
			pt_out^[pos_out] := 59;
		60: (* < detected *)
			IF pos_out > STRING_LENGTH - 4 THEN EXIT; END_IF;
			pt_out^[pos_out] := 38;
			pos_out := pos_out + 1;
			pt_out^[pos_out] := 108;
			pos_out := pos_out + 1;
			pt_out^[pos_out] := 116;
			pos_out := pos_out + 1;
			pt_out^[pos_out] := 59;
		62: (* > detected *)
			IF pos_out > STRING_LENGTH - 4 THEN EXIT; END_IF;
			pt_out^[pos_out] := 38;
			pos_out := pos_out + 1;
			pt_out^[pos_out] := 103;
			pos_out := pos_out + 1;
			pt_out^[pos_out] := 116;
			pos_out := pos_out + 1;
			pt_out^[pos_out] := 59;
	ELSE
		IF M AND B > 127 THEN
			tmp := CHARNAME(B);
			(* exit if output string has not enough space *)
			IF pos_out + LEN(tmp) + 2 <= 250 THEN
				pt_out^[pos_out] := 38;
				pos_out := pos_out + 1;
				FOR i := 1 TO LEN(tmp) DO
					pt_out^[pos_out] := CODE(tmp, i);
					pos_out := pos_out + 1;
				END_FOR;
				pt_out^[pos_out] := 59;
			END_IF;
		ELSE
			pt_out^[pos_out] := B;
		END_IF;
	END_CASE;
	(* increment in by 1 *)
	pos_in := pos_in + 1;
END_FOR;

(* terminate the output string *)
pt_out^[pos_out] := 0;



(* revision history
hm		3. mai. 2008	rev 1.0
	original version

hm		10. mai. 2008	rev 1.1
	stringlength 250
*)
END_FUNCTION

(* POU IP4_CHECK, ST *)
FUNCTION IP4_CHECK : BOOL
VAR_INPUT
	NIP : DWORD;
	LIP : DWORD;
	SM : DWORD;
END_VAR


(*
version 1.0	4. mar 2008
programmer 	hugo
tested by		oscat

IP4_CHECK testet ob eine Network IP und Local_IP im selben Subnet sind.

*)
IP4_CHECK := (NIP AND sm) = (LIP AND SM);


(* revision history
hm		4. mar 2008	rev 1.0
	original version

*)
END_FUNCTION

(* POU IRTRANS_RCV_1, ST *)
FUNCTION_BLOCK IRTRANS_RCV_1
VAR_INPUT CONSTANT
	DEV_CODE : STRING;
	KEY_CODE : STRING;
END_VAR
VAR_INPUT
	CMD : BOOL;
END_VAR
VAR_IN_OUT
	DEV : STRING;
	KEY : STRING;
END_VAR
VAR_OUTPUT
	Q : BOOL;
END_VAR


(*

version 1.3	06. dec. 2009
programmer 	hugo
tested BY	oscat

*)
Q := cmd AND dev_code = dev AND key_code = key;

(* revision history
hm	2. jan 2008		rev 1.0
	original version

hm	20. 6. 2008		rev 1.1
	performance improvement

hm	19. oct. 2008	rev 1.2
	changed input device_code to dev_code and device to dev for compatibility reasons

hm	06. dec. 2008	rev 1.3
	IRTRANS_1 renamed to IRTRANS_RCV_1

*)
END_FUNCTION_BLOCK

(* POU IRTRANS_RCV_8, ST *)
FUNCTION_BLOCK IRTRANS_RCV_8
VAR_INPUT CONSTANT
	dev_code : STRING;
	key_code_0 : STRING;
	key_code_1 : STRING;
	key_code_2 : STRING;
	key_code_3 : STRING;
	key_code_4 : STRING;
	key_code_5 : STRING;
	key_code_6 : STRING;
	key_code_7 : STRING;
END_VAR
VAR_INPUT
	CMD : BOOL;
END_VAR
VAR_IN_OUT
	DEV : STRING;
	KEY : STRING;
END_VAR
VAR_OUTPUT
	Q0, Q1, Q2, Q3, Q4, Q5, Q6, Q7 : BOOL;
END_VAR
VAR_TEMP
	decode: BOOL;
END_VAR

(*

version 1.3	06. dec. 2009
programmer 	hugo
tested BY	oscat

*)
decode := cmd AND dev_code = dev;

Q0 := key = key_code_0 AND decode;
Q1 := key = key_code_1 AND decode;
Q2 := key = key_code_2 AND decode;
Q3 := key = key_code_3 AND decode;
Q4 := key = key_code_4 AND decode;
Q5 := key = key_code_5 AND decode;
Q6 := key = key_code_6 AND decode;
Q7 := key = key_code_7 AND decode;


(* revision history
hm	2. jan 2008		rev 1.0
	original version

hm	17. oct 2008	rev 1.1
	improved performance

hm	19. oct. 2008	rev 1.2
	changed input device_code to dev_code and device to dev for compatibility reasons

hm	06. dec. 2008	rev 1.3
	IRTRANS_1 renamed to IRTRANS_RCV_8

*)
END_FUNCTION_BLOCK

(* POU IRTRANS_SND_1, ST *)
FUNCTION_BLOCK IRTRANS_SND_1
VAR_INPUT CONSTANT
	DEV_CODE : STRING;
	KEY_CODE : STRING;
END_VAR
VAR_INPUT
	IN : BOOL;
	T_REPEAT : TIME;
END_VAR
VAR_IN_OUT
	IP_C : IP_C; (* IP_Control Verwaltungsstruktur *)
	S_BUF : NETWORK_BUFFER_SHORT;
END_VAR
VAR_OUTPUT
	KEY : BYTE;
END_VAR
VAR
	skey : STRING;
	size : INT;
	str : STRING;
	t : TON;
	k : BYTE;
	lk : BYTE;
	d : BOOL;
END_VAR

(*
version 1.0		06. dec. 2009
programmer 		ks
tested by		ks
*)
d := IP_C.C_STATE > 127 AND (IP_C.MAILBOX[1] > 0 OR IP_C.C_MODE <> 5);
IF NOT d THEN RETURN; END_IF;

t(IN:= lk = k , PT:=T_REPEAT);

IF S_BUF.SIZE = 0 THEN
	IF IN THEN
		skey := KEY_CODE; k := 1;
	ELSE
		lk := 0;
		KEY := 0;
		RETURN; (* beenden wenn kein Key aktiv *)
	END_IF;

	IF lk <> k OR T.Q THEN (* anderer Key oder repeat wartezeit abgelaufen *)
		str := CONCAT('snd ',dev_code);
		str := CONCAT(str,',');
		str := CONCAT(str,skey);
		size := LEN(str);
		_STRING_TO_BUFFER(STR:=str, POS:=0, PT:=ADR(S_BUF.BUFFER), SIZE:=size);
		S_BUF.SIZE := size; (* Sendelänge eintragen *)
		KEY := k;
		lk := k; (* letzten Key speichern *)
		t(IN:=FALSE); (* Reset Time *)
	END_IF;
END_IF;

(* revision history
hm	6. dec 2009		rev 1.0
	original version
*)
END_FUNCTION_BLOCK

(* POU IRTRANS_SND_4, ST *)
FUNCTION_BLOCK IRTRANS_SND_4
VAR_INPUT CONSTANT
	DEV_CODE : STRING;
	KEY_CODE_0 : STRING;
	KEY_CODE_1 : STRING;
	KEY_CODE_2 : STRING;
	KEY_CODE_3 : STRING;
END_VAR
VAR_INPUT
	IN_0 : BOOL;
	IN_1 : BOOL;
	IN_2 : BOOL;
	IN_3 : BOOL;
	T_REPEAT : TIME;
END_VAR
VAR_IN_OUT
	IP_C : IP_C; (* IP_Control Verwaltungsstruktur *)
	S_BUF : NETWORK_BUFFER_SHORT;
END_VAR
VAR_OUTPUT
	KEY : BYTE;
END_VAR
VAR
	skey : STRING;
	size : INT;
	str : STRING;
	t : TON;
	k : BYTE;
	lk : BYTE;
	d : BOOL;
END_VAR

(*
version 1.0		06. dec. 2009
programmer 		ks
tested by		ks
*)
d := IP_C.C_STATE > 127 AND (IP_C.MAILBOX[1] > 0 OR IP_C.C_MODE <> 5);
IF NOT d THEN RETURN; END_IF;

t(IN:= lk = k , PT:=T_REPEAT);

IF S_BUF.SIZE = 0 THEN
	IF IN_0 THEN
		skey := KEY_CODE_0; k := 1;
	ELSIF IN_1 THEN
		skey := KEY_CODE_1; k := 2;
	ELSIF IN_2 THEN
		skey := KEY_CODE_2; k := 3;
	ELSIF IN_3 THEN
		skey := KEY_CODE_3; k := 4;
	ELSE
		lk := 0;
		KEY := 0;
		RETURN; (* beenden wenn kein Key aktiv *)
	END_IF;

	IF lk <> k OR T.Q THEN (* anderer Key oder repeat wartezeit abgelaufen *)
		str := CONCAT('snd ',dev_code);
		str := CONCAT(str,',');
		str := CONCAT(str,skey);
		size := LEN(str);
		_STRING_TO_BUFFER(STR:=str, POS:=0, PT:=ADR(S_BUF.BUFFER), SIZE:=size);
		S_BUF.SIZE := size; (* Sendelänge eintragen *)
		KEY := k;
		lk := k; (* letzten Key speichern *)
		t(IN:=FALSE); (* Reset Time *)
	END_IF;
END_IF;

(* revision history
hm	6. dec 2009		rev 1.0
	original version
*)
END_FUNCTION_BLOCK

(* POU IS_IP4, ST *)
FUNCTION IS_IP4 : BOOL
VAR_INPUT
	str : STRING;
END_VAR


(*
version 1.1	10. mar 2009
programmer 	kurt
tested by		hugo

IS_IP4 testet ob ein string eine gültige IPv4 Adresse enthält.

*)
IS_IP4 := COUNT_CHAR(str, 46) = 3;


(* revision history
hm	1. mar. 2008	rev 1.0
	original version

hm	10. mar. 2009	rev 1.1
	new code

*)
END_FUNCTION

(* POU IS_URLCHR, ST *)
FUNCTION IS_URLCHR : BOOL
VAR_INPUT
	IN : BYTE;
END_VAR


(*
version 1.0		27. apr. 2008
programmer 		hugo
tested by		hugo

IS_URL_CHR is true if a string contains only non reserved characters for an url.
the non reserved characters are : [A..Z], [a..z], [0..9], -_.~

*)
IS_URLCHR := ((IN > 47) AND (IN < 58)) OR ((IN > 64) AND (IN < 91)) OR ((IN > 96) AND (IN < 123)) OR (in = 126) OR (in = 95) OR (in =45) OR (in =46);


(* revision history
hm		27. apr. 2008	rev 1.0
	original version

*)
END_FUNCTION

(* POU TN_SC_READ_ATTR, ST *)
FUNCTION_BLOCK TN_SC_READ_ATTR
VAR
	in_Offset : INT;
END_VAR
VAR_INPUT
	Iin_Y : INT;
	Iin_X : INT;
END_VAR
VAR_OUTPUT
	Oby_ATTR : BYTE;
END_VAR
VAR_IN_OUT
	Xus_TN_SCREEN : us_TN_SCREEN;
END_VAR

(*
version 1.0		10. mai 2010
programmer		ks
tested by		ks

TN_SC_READ_ATTR gibt den Farbcode einer Koordinate vom Bildschirm aus

*)
IF TN_SC_XY_ERROR(Iin_X,Iin_Y) THEN RETURN; END_IF;
in_Offset := (Iin_Y * 80) + Iin_X;
Oby_ATTR := Xus_TN_SCREEN.bya_COLOR[in_Offset]; (* Attribute auslesen *)

(* revision history
ks	10. mai. 2010	rev 1.0
	original version
*)
END_FUNCTION_BLOCK

(* POU TN_SC_READ_CHAR, ST *)
FUNCTION_BLOCK TN_SC_READ_CHAR
VAR
	in_Offset : INT;
END_VAR
VAR_INPUT
	Iin_Y : INT;
	Iin_X : INT;
END_VAR
VAR_OUTPUT
	Oby_CHAR : BYTE;
END_VAR
VAR_IN_OUT
	Xus_TN_SCREEN : us_TN_SCREEN;
END_VAR

(*
version 1.0		10. mai 2010
programmer		ks
tested by		ks

TN_SC_READ_CHAR gibt das Zeichen einer Koordinate vom Bildschirm aus
*)
IF TN_SC_XY_ERROR(Iin_X,Iin_Y) THEN RETURN; END_IF;
in_Offset := (Iin_Y * 80) + Iin_X;
Oby_CHAR := Xus_TN_SCREEN.bya_CHAR[in_Offset]; (* Charakter auslesen *)

(* revision history
ks	10. mai. 2010	rev 1.0
	original version
*)
END_FUNCTION_BLOCK

(* POU TN_SC_WRITE_ATTR, ST *)
FUNCTION_BLOCK TN_SC_WRITE_ATTR
VAR
	in_Offset : INT;
END_VAR
VAR_INPUT
	Iin_Y : INT;
	Iin_X : INT;
	Iby_ATTR : BYTE;
END_VAR
VAR_IN_OUT
	Xus_TN_SCREEN : us_TN_SCREEN;
END_VAR

(*
version 1.0		10. mai 2010
programmer		ks
tested by		ks

TN_SC_WRITE_ATTR ändert an der angegebenen Koordinate den Farbcode
*)
IF TN_SC_XY_ERROR(Iin_X,Iin_Y) THEN RETURN; END_IF;
in_Offset := (Iin_Y * 80) + Iin_X;
Xus_TN_SCREEN.bya_COLOR[in_Offset] := Iby_ATTR; (* Attribute schreiben *)

(* revision history
ks	10. mai. 2010	rev 1.0
	original version
*)
END_FUNCTION_BLOCK

(* POU TN_SC_WRITE_CHAR, ST *)
FUNCTION_BLOCK TN_SC_WRITE_CHAR
VAR
	in_Offset : INT;
END_VAR
VAR_INPUT
	Iin_Y : INT;
	Iin_X : INT;
	Iby_CHAR : BYTE;
END_VAR
VAR_IN_OUT
	Xus_TN_SCREEN : us_TN_SCREEN;
END_VAR

(*
version 1.0		10. mai 2010
programmer		ks
tested by		ks

TN_SC_WRITE_CHAR schreibt ein einzelnes Zeichen an die angegebenen Koordinate ohne den vorhandenen Farbcode zu ändern 
*)
IF TN_SC_XY_ERROR(Iin_X,Iin_Y) THEN RETURN; END_IF;
in_Offset := (Iin_Y * 80) + Iin_X;
Xus_TN_SCREEN.bya_CHAR[in_Offset] := Iby_CHAR; (* Charakter schreiben *)

(* revision history
ks	10. mai. 2010	rev 1.0
	original version
*)
END_FUNCTION_BLOCK

(* POU TN_SC_WRITE_EOS, ST *)
FUNCTION_BLOCK TN_SC_WRITE_EOS
VAR
	TN_SC_WRITE : TN_SC_WRITE;
END_VAR
VAR_INPUT
	Iby_ATTR : BYTE;
	Ist_STRING : STRING;
END_VAR
VAR_IN_OUT
	Xus_TN_SCREEN : us_TN_SCREEN;
END_VAR

(*
version 1.0		10. mai 2010
programmer		ks
tested by		ks

TN_SC_WRITE_EOS schreibt einem Text an das Ende des zuletzt geschreibene Texts 
*)
TN_SC_WRITE(Iin_Y := Xus_TN_SCREEN.in_EOS_Offset / 80, (* aktuelle Zeile ausrechnen *)
			Iin_X := Xus_TN_SCREEN.in_EOS_Offset MOD 80, (* aktuelle Spalte ausrechnen *)
			Iby_ATTR := Iby_ATTR,
			Ist_STRING := Ist_STRING,
			Xus_TN_SCREEN := Xus_TN_SCREEN);

(* revision history
ks	10. mai. 2010	rev 1.0
	original version
*)
END_FUNCTION_BLOCK

(* POU URL_DECODE, ST *)
FUNCTION URL_DECODE : STRING(STRING_LENGTH)
VAR_INPUT
	IN : STRING(STRING_LENGTH);
END_VAR
VAR
	pos : INT;
	seq : STRING(3);
	new : STRING(1);
END_VAR


(*
version 1.2		10. may. 2010
programmer 	hugo
tested by		hugo

URL_DECODE checks a string if it contains non reserved characters represented by a % followed with the two digit hex code and converts them to their ascii code.
the non reserved characters are : [A..Z], [a..z], [0..9], -_.~
for example the character sequence '%23' will be converted to '#'.

*)
URL_DECODE := IN;
pos := FIND(URL_DECODE,'%');
WHILE pos > 0 DO
	seq := MID(URL_DECODE,2,pos + 1);
	new := CHR_TO_STRING(DWORD_TO_BYTE(HEX_TO_DWORD(seq)));
	URL_DECODE := REPLACE(URL_DECODE, new, 3, pos);
	pos := FIND(URL_DECODE,'%');
END_WHILE;


(* revision history
hm	27. apr. 2008	rev 1.0
	original version

hm	17. dec. 2008	rev 1.1
	changes name of function chr to chr_to_string

ks	10. mai. 2008	rev 1.2
	stringlength 250
*)
END_FUNCTION

(* POU URL_ENCODE, ST *)
FUNCTION URL_ENCODE : STRING(STRING_LENGTH)
VAR_INPUT
	IN : STRING(STRING_LENGTH);
END_VAR
VAR
	pt_in : POINTER TO ARRAY[1..255] OF BYTE;
	pt_out : POINTER TO ARRAY[1..256] OF BYTE;
	pos_in : INT;
	pos_out : INT;
	stop : INT;
	tb : BYTE;
END_VAR


(*
version 1.1		10. may. 2010
programmer 	hugo
tested by		hugo

URL_ENCODE checks a string if it contains only non reserved characters for an url.
the non reserved characters are : [A..Z], [a..z], [0..9], -_.~
if reserved characters are found then these characters are converted to %HH while HH is the Hexadezimal representation of the character in Alphabetic Letters.
for example the reserved character # will be converted to '%23'.

*)
pt_in  := ADR(in);
pt_out := ADR(URL_ENCODE);

(* scan the input string and convert unallowed characters *)
pos_in := 1;
stop := LEN(in);
FOR pos_out := 1 TO 250 DO
	IF pos_in > stop THEN
		EXIT;
	ELSIF IS_URLCHR(pt_in^[pos_in]) THEN
		pt_out^[pos_out] := pt_in^[pos_in];
		(* increment in by 1 *)
		pos_in := pos_in + 1;
	ELSE
		(* cannot fit 3 digits, exit *)
		IF pos_out > 248 THEN EXIT; END_IF;
		(* invalid character that needs to be converted *)
		pt_out^[pos_out] := 37;    (* start with % sign *)
		pos_out := pos_out + 1;
		(* need to add the two hex digits *)
		tb := SHR(pt_in^[pos_in],4);
		IF tb > 9 THEN
			pt_out^[pos_out] := tb + 55;
		ELSE
			pt_out^[pos_out] := tb + 48;
		END_IF;
		pos_out := pos_out + 1;
		tb := pt_in^[pos_in] AND 16#0F;
		IF tb > 9 THEN
			pt_out^[pos_out] := tb + 55;
		ELSE
			pt_out^[pos_out] := tb + 48;
		END_IF;
		(* increment in and out because out has to move 3 digits *)
		pos_in := pos_in + 1;
	END_IF;
END_FOR;

(* terminate the output string *)
pt_out^[pos_out] := 0;

(* revision history
hm	27. apr. 2008	rev 1.0
	original version

ks	10. mai. 2008	rev 1.1
	stringlength 250

*)
END_FUNCTION

(* POU URL_TO_STRING, ST *)
FUNCTION URL_TO_STRING : STRING(STRING_LENGTH)
VAR_INPUT
	IN : URL;
END_VAR


(*
version 1.1		10. may. 2010
programmer 	hugo
tested by		oscat

URL_TO_STRING generates a string from URL information suppied in IN..

*)
(*

http://hans:geheim@www.example.org:80/demo/example.cgi?land=de&stadt=aa#abschnitt1
|         |         |                  |                                |   |                                    |                                    |
|         |         |                 Host                         |   Pfad                            Query                           Anker
|         |         Passwort                                  Port
|        Benutzer
Protokoll

*)

(* attach protocol *)
IF IN.PROTOCOL <> '' THEN URL_TO_STRING := CONCAT(IN.PROTOCOL,'://'); END_IF;

(* attach user and password *)
IF IN.USER <> '' THEN
	URL_TO_STRING := CONCAT(URL_TO_STRING, IN.USER);
	IF IN.PASSWORD <> '' THEN
		URL_TO_STRING := CONCAT(URL_TO_STRING, ':');
		URL_TO_STRING := CONCAT(URL_TO_STRING, IN.PASSWORD);
	END_IF;
	URL_TO_STRING := CONCAT(URL_TO_STRING, '@');
END_IF;

(* attach domain *)
URL_TO_STRING := CONCAT(URL_TO_STRING, IN.DOMAIN);

(* attach Port *)
IF IN.PORT > 0 THEN
	URL_TO_STRING := CONCAT(URL_TO_STRING, ':');
	URL_TO_STRING := CONCAT(URL_TO_STRING, WORD_TO_STRING(IN.PORT));
END_IF;

(* attach path *)
URL_TO_STRING := CONCAT(URL_TO_STRING, IN.PATH);

(* attach query *)
IF IN.QUERY <> '' THEN
	URL_TO_STRING := CONCAT(URL_TO_STRING, '?');
	URL_TO_STRING := CONCAT(URL_TO_STRING, IN.QUERY);
END_IF;

(* attach anchor *)
IF IN.ANCHOR <> '' THEN
	URL_TO_STRING := CONCAT(URL_TO_STRING, '#');
	URL_TO_STRING := CONCAT(URL_TO_STRING, IN.ANCHOR);
END_IF;

(* revision history
hm	18. apr 2008	rev 1.0
	original version

ks	10. mai. 2008	rev 1.1
	stringlength 250
*)
END_FUNCTION
